SPLINE
SPL {X  -160.000, Y  +499.279, Z    +0.000, E1   +38.981, E3 +82505.209}
SPL {X  -160.000, Y  +490.068, Z    +0.000, E1   +40.198, E3 +82521.513}
SPL {X  -160.000, Y  +481.368, Z    +0.000, E1   +41.274, E3 +82536.503}
SPL {X  -160.000, Y  +470.910, Z    +0.000, E1   +42.658, E3 +82553.012}
SPL {X  -160.000, Y  +460.219, Z    +0.000, E1   +43.912, E3 +82569.633}
SPL {X  -160.000, Y  +451.951, Z    +0.000, E1   +44.355, E3 +82585.198}
SPL {X  -160.000, Y  +442.331, Z    +0.000, E1   +44.390, E3 +82606.062}
SPL {X  -160.000, Y  +433.037, Z    +0.000, E1   +44.348, E3 +82626.336}
SPL {X  -160.000, Y  +424.435, Z    +0.000, E1   +44.358, E3 +82645.005}
SPL {X  -160.000, Y  +416.015, Z    +0.000, E1   +44.348, E3 +82663.325}
SPL {X  -160.000, Y  +407.167, Z    +0.000, E1   +44.365, E3 +82682.535}
SPL {X  -160.000, Y  +397.599, Z    +0.000, E1   +44.371, E3 +82703.344}
SPL {X  -160.000, Y  +388.533, Z    +0.000, E1   +44.340, E3 +82723.119}
SPL {X  -159.759, Y  +380.021, Z    +0.000, E1   +44.311, E3 +82741.851}
SPL {X  -159.014, Y  +371.065, Z    +0.000, E1   +44.193, E3 +82762.089}
SPL {X  -157.745, Y  +362.030, Z    +0.000, E1   +43.965, E3 +82783.071}
SPL {X  -156.258, Y  +354.400, Z    +0.000, E1   +43.653, E3 +82801.278}
SPL {X  -154.385, Y  +346.786, Z    +0.000, E1   +43.356, E3 +82819.690}
SPL {X  -152.146, Y  +339.286, Z    +0.000, E1   +42.904, E3 +82838.324}
SPL {X  -149.854, Y  +332.731, Z    +0.000, E1   +42.474, E3 +82854.852}
SPL {X  -145.635, Y  +322.541, Z    +0.000, E1   +36.397, E3 +82930.811}
ENDSPLINE

SPLINE
SPL {X  -156.682, Y  +356.385, Z    +0.000, E1   +19.033, E3 +82989.117}
SPL {X  -159.526, Y  +376.492, Z    +0.000, E1    +8.067, E3 +82999.026}
SPL {X  -159.961, Y  +385.275, Z    +0.000, E1    +2.550, E3 +83001.065}
SPL {X  -160.000, Y  +390.345, Z    +0.000, E1    -1.188, E3 +83001.791}
SPL {X  -160.000, Y  +395.838, Z    +0.000, E1    -6.211, E3 +83002.734}
SPL {X  -160.000, Y  +403.277, Z    +0.000, E1   -14.057, E3 +83004.685}
SPL {X  -160.000, Y  +414.316, Z    +0.000, E1   -24.810, E3 +83009.758}
SPL {X  -160.000, Y  +442.604, Z    +0.000, E1   -40.161, E3 +83031.893}
SPL {X  -160.000, Y  +482.867, Z    +0.000, E1   -45.148, E3 +83092.109}
SPL {X  -160.000, Y  +494.769, Z    +0.000, E1   -45.151, E3 +83117.328}
SPL {X  -160.000, Y  +505.761, Z    +0.000, E1   -45.118, E3 +83140.642}
SPL {X  -160.000, Y  +517.347, Z    +0.000, E1   -45.173, E3 +83165.080}
SPL {X  -160.000, Y  +529.298, Z    +0.000, E1   -45.138, E3 +83190.463}
SPL {X  -160.000, Y  +540.664, Z    +0.000, E1   -45.139, E3 +83214.541}
SPL {X  -160.000, Y  +552.011, Z    +0.000, E1   -45.139, E3 +83238.577}
SPL {X  -160.000, Y  +563.667, Z    +0.000, E1   -45.146, E3 +83263.257}
SPL {X  -160.000, Y  +574.965, Z    +0.000, E1   -45.125, E3 +83287.233}
SPL {X  -160.000, Y  +585.644, Z    +0.000, E1   -45.117, E3 +83309.873}
SPL {X  -160.000, Y  +596.819, Z    +0.000, E1   -45.144, E3 +83333.514}
SPL {X  -160.000, Y  +608.165, Z    +0.000, E1   -45.120, E3 +83357.589}
SPL {X  -160.000, Y  +619.270, Z    +0.000, E1   -45.132, E3 +83381.091}
SPL {X  -160.000, Y  +629.968, Z    +0.000, E1   -45.117, E3 +83403.758}
SPL {X  -160.000, Y  +640.750, Z    +0.000, E1   -45.131, E3 +83426.581}
SPL {X  -160.000, Y  +651.429, Z    +0.000, E1   -45.117, E3 +83449.222}
SPL {X  -160.000, Y  +662.434, Z    +0.000, E1   -45.129, E3 +83472.566}
SPL {X  -159.992, Y  +673.110, Z    +0.000, E1   -45.097, E3 +83495.258}
SPL {X  -159.521, Y  +683.874, Z    +0.000, E1   -45.054, E3 +83518.514}
SPL {X  -158.435, Y  +693.823, Z    +0.000, E1   -44.810, E3 +83540.818}
SPL {X  -156.807, Y  +703.304, Z    +0.000, E1   -44.558, E3 +83562.539}
SPL {X  -154.802, Y  +711.950, Z    +0.000, E1   -44.141, E3 +83582.999}
SPL {X  -152.641, Y  +719.464, Z    +0.000, E1   -43.749, E3 +83601.114}
SPL {X  -149.826, Y  +727.645, Z    +0.000, E1   -43.252, E3 +83621.217}
SPL {X  -145.307, Y  +738.478, Z    +0.000, E1   -36.676, E3 +83701.285}
ENDSPLINE

SPLINE
SPL {X  -155.601, Y  +708.762, Z    +0.000, E1   -21.463, E3 +83756.072}
SPL {X  -158.549, Y  +693.002, Z    +0.000, E1   -13.406, E3 +83765.062}
SPL {X  -159.716, Y  +681.031, Z    +0.000, E1    -6.529, E3 +83769.212}
SPL {X  -160.000, Y  +671.641, Z    +0.000, E1    -0.547, E3 +83770.929}
SPL {X  -160.000, Y  +665.424, Z    +0.000, E1    +5.044, E3 +83771.877}
SPL {X  -160.000, Y  +658.015, Z    +0.000, E1   +12.630, E3 +83773.795}
SPL {X  -160.000, Y  +645.110, Z    +0.000, E1   +25.142, E3 +83779.595}
SPL {X  -160.000, Y  +611.664, Z    +0.000, E1   +41.262, E3 +83809.324}
SPL {X  -160.000, Y  +581.433, Z    +0.000, E1   +44.103, E3 +83859.061}
SPL {X  -160.000, Y  +572.090, Z    +0.000, E1   +44.120, E3 +83879.526}
SPL {X  -160.000, Y  +563.431, Z    +0.000, E1   +44.084, E3 +83898.579}
SPL {X  -160.000, Y  +556.107, Z    +0.000, E1   +44.076, E3 +83914.647}
SPL {X  -160.000, Y  +549.181, Z    +0.000, E1   +44.079, E3 +83929.807}
SPL {X  -160.000, Y  +542.413, Z    +0.000, E1   +44.088, E3 +83944.641}
SPL {X  -160.000, Y  +534.609, Z    +0.000, E1   +44.095, E3 +83961.751}
SPL {X  -160.000, Y  +527.457, Z    +0.000, E1   +44.070, E3 +83977.461}
SPL {X  -160.000, Y  +520.912, Z    +0.000, E1   +44.079, E3 +83991.802}
SPL {X  -160.000, Y  +514.086, Z    +0.000, E1   +44.081, E3 +84006.750}
SPL {X  -160.000, Y  +507.208, Z    +0.000, E1   +44.082, E3 +84021.827}
SPL {X  -160.000, Y  +499.184, Z    +0.000, E1   +44.113, E3 +84039.385}
ENDSPLINE

SPLINE
SPL {X  -160.000, Y  +503.824, Z    +0.000, E1   +39.488, E3 +84055.434}
ENDSPLINE

SPLINE
SPL {X  -160.000, Y  +499.279, Z    +0.000, E1   +38.981, E3 +84070.424}
SPL {X  -160.000, Y  +490.068, Z    +0.000, E1   +40.198, E3 +84086.728}
SPL {X  -160.000, Y  +481.368, Z    +0.000, E1   +41.274, E3 +84101.717}
SPL {X  -160.000, Y  +470.910, Z    +0.000, E1   +42.658, E3 +84118.226}
SPL {X  -160.000, Y  +460.219, Z    +0.000, E1   +43.912, E3 +84134.847}
SPL {X  -160.000, Y  +451.951, Z    +0.000, E1   +44.355, E3 +84150.412}
SPL {X  -160.000, Y  +442.331, Z    +0.000, E1   +44.390, E3 +84171.276}
SPL {X  -160.000, Y  +433.037, Z    +0.000, E1   +44.348, E3 +84191.550}
SPL {X  -160.000, Y  +424.435, Z    +0.000, E1   +44.358, E3 +84210.219}
SPL {X  -160.000, Y  +416.015, Z    +0.000, E1   +44.348, E3 +84228.539}
SPL {X  -160.000, Y  +407.167, Z    +0.000, E1   +44.365, E3 +84247.750}
SPL {X  -160.000, Y  +397.599, Z    +0.000, E1   +44.371, E3 +84268.558}
SPL {X  -160.000, Y  +388.533, Z    +0.000, E1   +44.340, E3 +84288.333}
SPL {X  -159.759, Y  +380.021, Z    +0.000, E1   +44.311, E3 +84307.065}
SPL {X  -159.014, Y  +371.065, Z    +0.000, E1   +44.193, E3 +84327.303}
SPL {X  -157.745, Y  +362.030, Z    +0.000, E1   +43.965, E3 +84348.285}
SPL {X  -156.258, Y  +354.400, Z    +0.000, E1   +43.653, E3 +84366.492}
SPL {X  -154.385, Y  +346.786, Z    +0.000, E1   +43.356, E3 +84384.904}
SPL {X  -152.146, Y  +339.286, Z    +0.000, E1   +42.904, E3 +84403.539}
SPL {X  -149.854, Y  +332.731, Z    +0.000, E1   +42.474, E3 +84420.066}
SPL {X  -145.635, Y  +322.541, Z    +0.000, E1   +36.397, E3 +84496.025}
ENDSPLINE

SPLINE
SPL {X  -156.682, Y  +356.385, Z    +0.000, E1   +19.033, E3 +84554.331}
SPL {X  -159.526, Y  +376.492, Z    +0.000, E1    +8.067, E3 +84564.241}
SPL {X  -159.961, Y  +385.275, Z    +0.000, E1    +2.550, E3 +84566.279}
SPL {X  -160.000, Y  +390.345, Z    +0.000, E1    -1.188, E3 +84567.005}
SPL {X  -160.000, Y  +395.838, Z    +0.000, E1    -6.211, E3 +84567.948}
SPL {X  -160.000, Y  +403.277, Z    +0.000, E1   -14.057, E3 +84569.900}
SPL {X  -160.000, Y  +414.316, Z    +0.000, E1   -24.810, E3 +84574.973}
SPL {X  -160.000, Y  +442.604, Z    +0.000, E1   -40.161, E3 +84597.107}
SPL {X  -160.000, Y  +482.867, Z    +0.000, E1   -45.148, E3 +84657.323}
SPL {X  -160.000, Y  +494.769, Z    +0.000, E1   -45.151, E3 +84682.542}
SPL {X  -160.000, Y  +505.761, Z    +0.000, E1   -45.118, E3 +84705.856}
SPL {X  -160.000, Y  +517.347, Z    +0.000, E1   -45.173, E3 +84730.294}
SPL {X  -160.000, Y  +529.298, Z    +0.000, E1   -45.138, E3 +84755.677}
SPL {X  -160.000, Y  +540.664, Z    +0.000, E1   -45.139, E3 +84779.755}
SPL {X  -160.000, Y  +552.011, Z    +0.000, E1   -45.139, E3 +84803.791}
SPL {X  -160.000, Y  +563.667, Z    +0.000, E1   -45.146, E3 +84828.471}
SPL {X  -160.000, Y  +574.965, Z    +0.000, E1   -45.125, E3 +84852.447}
SPL {X  -160.000, Y  +585.644, Z    +0.000, E1   -45.117, E3 +84875.087}
SPL {X  -160.000, Y  +596.819, Z    +0.000, E1   -45.144, E3 +84898.729}
SPL {X  -160.000, Y  +608.165, Z    +0.000, E1   -45.120, E3 +84922.803}
SPL {X  -160.000, Y  +619.270, Z    +0.000, E1   -45.132, E3 +84946.305}
SPL {X  -160.000, Y  +629.968, Z    +0.000, E1   -45.117, E3 +84968.972}
SPL {X  -160.000, Y  +640.750, Z    +0.000, E1   -45.131, E3 +84991.795}
SPL {X  -160.000, Y  +651.429, Z    +0.000, E1   -45.117, E3 +85014.436}
SPL {X  -160.000, Y  +662.434, Z    +0.000, E1   -45.129, E3 +85037.780}
SPL {X  -159.992, Y  +673.110, Z    +0.000, E1   -45.097, E3 +85060.473}
SPL {X  -159.521, Y  +683.874, Z    +0.000, E1   -45.054, E3 +85083.728}
SPL {X  -158.435, Y  +693.823, Z    +0.000, E1   -44.810, E3 +85106.032}
SPL {X  -156.807, Y  +703.304, Z    +0.000, E1   -44.558, E3 +85127.753}
SPL {X  -154.802, Y  +711.950, Z    +0.000, E1   -44.141, E3 +85148.213}
SPL {X  -152.641, Y  +719.464, Z    +0.000, E1   -43.749, E3 +85166.329}
SPL {X  -149.826, Y  +727.645, Z    +0.000, E1   -43.252, E3 +85186.431}
SPL {X  -145.307, Y  +738.478, Z    +0.000, E1   -36.676, E3 +85266.499}
ENDSPLINE

SPLINE
SPL {X  -155.601, Y  +708.762, Z    +0.000, E1   -21.463, E3 +85321.286}
SPL {X  -158.549, Y  +693.002, Z    +0.000, E1   -13.406, E3 +85330.276}
SPL {X  -159.716, Y  +681.031, Z    +0.000, E1    -6.529, E3 +85334.427}
SPL {X  -160.000, Y  +671.641, Z    +0.000, E1    -0.547, E3 +85336.143}
SPL {X  -160.000, Y  +665.424, Z    +0.000, E1    +5.044, E3 +85337.091}
SPL {X  -160.000, Y  +658.015, Z    +0.000, E1   +12.630, E3 +85339.009}
SPL {X  -160.000, Y  +645.110, Z    +0.000, E1   +25.142, E3 +85344.809}
SPL {X  -160.000, Y  +611.664, Z    +0.000, E1   +41.262, E3 +85374.539}
SPL {X  -160.000, Y  +581.433, Z    +0.000, E1   +44.103, E3 +85424.275}
SPL {X  -160.000, Y  +572.090, Z    +0.000, E1   +44.120, E3 +85444.740}
SPL {X  -160.000, Y  +563.431, Z    +0.000, E1   +44.084, E3 +85463.793}
SPL {X  -160.000, Y  +556.107, Z    +0.000, E1   +44.076, E3 +85479.861}
SPL {X  -160.000, Y  +549.181, Z    +0.000, E1   +44.079, E3 +85495.021}
SPL {X  -160.000, Y  +542.413, Z    +0.000, E1   +44.088, E3 +85509.855}
SPL {X  -160.000, Y  +534.609, Z    +0.000, E1   +44.095, E3 +85526.965}
SPL {X  -160.000, Y  +527.457, Z    +0.000, E1   +44.070, E3 +85542.675}
SPL {X  -160.000, Y  +520.912, Z    +0.000, E1   +44.079, E3 +85557.016}
SPL {X  -160.000, Y  +514.086, Z    +0.000, E1   +44.081, E3 +85571.964}
SPL {X  -160.000, Y  +507.208, Z    +0.000, E1   +44.082, E3 +85587.041}
SPL {X  -160.000, Y  +499.184, Z    +0.000, E1   +44.113, E3 +85604.599}
ENDSPLINE

SPLINE
SPL {X  -160.000, Y  +503.824, Z    +0.000, E1   +39.488, E3 +85620.648}
ENDSPLINE

SPLINE
SPL {X  -160.000, Y  +499.279, Z    +0.000, E1   +38.981, E3 +85635.638}
SPL {X  -160.000, Y  +490.068, Z    +0.000, E1   +40.198, E3 +85651.942}
SPL {X  -160.000, Y  +481.368, Z    +0.000, E1   +41.274, E3 +85666.932}
SPL {X  -160.000, Y  +470.910, Z    +0.000, E1   +42.658, E3 +85683.440}
SPL {X  -160.000, Y  +460.219, Z    +0.000, E1   +43.912, E3 +85700.061}
SPL {X  -160.000, Y  +451.951, Z    +0.000, E1   +44.355, E3 +85715.626}
SPL {X  -160.000, Y  +442.331, Z    +0.000, E1   +44.390, E3 +85736.491}
SPL {X  -160.000, Y  +433.037, Z    +0.000, E1   +44.348, E3 +85756.765}
SPL {X  -160.000, Y  +424.435, Z    +0.000, E1   +44.358, E3 +85775.433}
SPL {X  -160.000, Y  +416.015, Z    +0.000, E1   +44.348, E3 +85793.753}
SPL {X  -160.000, Y  +407.167, Z    +0.000, E1   +44.365, E3 +85812.964}
SPL {X  -160.000, Y  +397.599, Z    +0.000, E1   +44.371, E3 +85833.772}
SPL {X  -160.000, Y  +388.533, Z    +0.000, E1   +44.340, E3 +85853.547}
SPL {X  -159.759, Y  +380.021, Z    +0.000, E1   +44.311, E3 +85872.279}
SPL {X  -159.014, Y  +371.065, Z    +0.000, E1   +44.193, E3 +85892.517}
SPL {X  -157.745, Y  +362.030, Z    +0.000, E1   +43.965, E3 +85913.499}
SPL {X  -156.258, Y  +354.400, Z    +0.000, E1   +43.653, E3 +85931.706}
SPL {X  -154.385, Y  +346.786, Z    +0.000, E1   +43.356, E3 +85950.118}
SPL {X  -152.146, Y  +339.286, Z    +0.000, E1   +42.904, E3 +85968.753}
SPL {X  -149.854, Y  +332.731, Z    +0.000, E1   +42.474, E3 +85985.281}
SPL {X  -145.635, Y  +322.541, Z    +0.000, E1   +36.397, E3 +86061.240}
ENDSPLINE

SPLINE
SPL {X  -156.682, Y  +356.385, Z    +0.000, E1   +19.033, E3 +86119.546}
SPL {X  -159.526, Y  +376.492, Z    +0.000, E1    +8.067, E3 +86129.455}
SPL {X  -159.961, Y  +385.275, Z    +0.000, E1    +2.550, E3 +86131.493}
SPL {X  -160.000, Y  +390.345, Z    +0.000, E1    -1.188, E3 +86132.219}
SPL {X  -160.000, Y  +395.838, Z    +0.000, E1    -6.211, E3 +86133.163}
SPL {X  -160.000, Y  +403.277, Z    +0.000, E1   -14.057, E3 +86135.114}
SPL {X  -160.000, Y  +414.316, Z    +0.000, E1   -24.810, E3 +86140.187}
SPL {X  -160.000, Y  +442.604, Z    +0.000, E1   -40.161, E3 +86162.321}
SPL {X  -160.000, Y  +482.867, Z    +0.000, E1   -45.148, E3 +86222.537}
SPL {X  -160.000, Y  +494.769, Z    +0.000, E1   -45.151, E3 +86247.756}
SPL {X  -160.000, Y  +505.761, Z    +0.000, E1   -45.118, E3 +86271.070}
SPL {X  -160.000, Y  +517.347, Z    +0.000, E1   -45.173, E3 +86295.508}
SPL {X  -160.000, Y  +529.298, Z    +0.000, E1   -45.138, E3 +86320.891}
SPL {X  -160.000, Y  +540.664, Z    +0.000, E1   -45.139, E3 +86344.969}
SPL {X  -160.000, Y  +552.011, Z    +0.000, E1   -45.139, E3 +86369.005}
SPL {X  -160.000, Y  +563.667, Z    +0.000, E1   -45.146, E3 +86393.685}
SPL {X  -160.000, Y  +574.965, Z    +0.000, E1   -45.125, E3 +86417.661}
SPL {X  -160.000, Y  +585.644, Z    +0.000, E1   -45.117, E3 +86440.301}
SPL {X  -160.000, Y  +596.819, Z    +0.000, E1   -45.144, E3 +86463.943}
SPL {X  -160.000, Y  +608.165, Z    +0.000, E1   -45.120, E3 +86488.017}
SPL {X  -160.000, Y  +619.270, Z    +0.000, E1   -45.132, E3 +86511.520}
SPL {X  -160.000, Y  +629.968, Z    +0.000, E1   -45.117, E3 +86534.186}
SPL {X  -160.000, Y  +640.750, Z    +0.000, E1   -45.131, E3 +86557.009}
SPL {X  -160.000, Y  +651.429, Z    +0.000, E1   -45.117, E3 +86579.650}
SPL {X  -160.000, Y  +662.434, Z    +0.000, E1   -45.129, E3 +86602.994}
SPL {X  -159.992, Y  +673.110, Z    +0.000, E1   -45.097, E3 +86625.687}
SPL {X  -159.521, Y  +683.874, Z    +0.000, E1   -45.054, E3 +86648.942}
SPL {X  -158.435, Y  +693.823, Z    +0.000, E1   -44.810, E3 +86671.246}
SPL {X  -156.807, Y  +703.304, Z    +0.000, E1   -44.558, E3 +86692.967}
SPL {X  -154.802, Y  +711.950, Z    +0.000, E1   -44.141, E3 +86713.427}
SPL {X  -152.641, Y  +719.464, Z    +0.000, E1   -43.749, E3 +86731.543}
SPL {X  -149.826, Y  +727.645, Z    +0.000, E1   -43.252, E3 +86751.646}
SPL {X  -145.307, Y  +738.478, Z    +0.000, E1   -36.676, E3 +86831.713}
ENDSPLINE

SPLINE
SPL {X  -155.601, Y  +708.762, Z    +0.000, E1   -21.463, E3 +86886.500}
SPL {X  -158.549, Y  +693.002, Z    +0.000, E1   -13.406, E3 +86895.491}
SPL {X  -159.716, Y  +681.031, Z    +0.000, E1    -6.529, E3 +86899.641}
SPL {X  -160.000, Y  +671.641, Z    +0.000, E1    -0.547, E3 +86901.357}
SPL {X  -160.000, Y  +665.424, Z    +0.000, E1    +5.044, E3 +86902.306}
SPL {X  -160.000, Y  +658.015, Z    +0.000, E1   +12.630, E3 +86904.223}
SPL {X  -160.000, Y  +645.110, Z    +0.000, E1   +25.142, E3 +86910.023}
SPL {X  -160.000, Y  +611.664, Z    +0.000, E1   +41.262, E3 +86939.753}
SPL {X  -160.000, Y  +581.433, Z    +0.000, E1   +44.103, E3 +86989.489}
SPL {X  -160.000, Y  +572.090, Z    +0.000, E1   +44.120, E3 +87009.954}
SPL {X  -160.000, Y  +563.431, Z    +0.000, E1   +44.084, E3 +87029.007}
SPL {X  -160.000, Y  +556.107, Z    +0.000, E1   +44.076, E3 +87045.075}
SPL {X  -160.000, Y  +549.181, Z    +0.000, E1   +44.079, E3 +87060.235}
SPL {X  -160.000, Y  +542.413, Z    +0.000, E1   +44.088, E3 +87075.069}
SPL {X  -160.000, Y  +534.609, Z    +0.000, E1   +44.095, E3 +87092.179}
SPL {X  -160.000, Y  +527.457, Z    +0.000, E1   +44.070, E3 +87107.889}
SPL {X  -160.000, Y  +520.912, Z    +0.000, E1   +44.079, E3 +87122.230}
SPL {X  -160.000, Y  +514.086, Z    +0.000, E1   +44.081, E3 +87137.179}
SPL {X  -160.000, Y  +507.208, Z    +0.000, E1   +44.082, E3 +87152.255}
SPL {X  -160.000, Y  +499.184, Z    +0.000, E1   +44.113, E3 +87169.813}
ENDSPLINE

SPLINE
SPL {X  -160.000, Y  +503.824, Z    +0.000, E1   +39.488, E3 +87185.862}
ENDSPLINE

SPLINE
SPL {X  -160.000, Y  +499.279, Z    +0.000, E1   +38.981, E3 +87200.852}
SPL {X  -160.000, Y  +490.068, Z    +0.000, E1   +40.198, E3 +87217.156}
SPL {X  -160.000, Y  +481.368, Z    +0.000, E1   +41.274, E3 +87232.146}
SPL {X  -160.000, Y  +470.910, Z    +0.000, E1   +42.658, E3 +87248.654}
SPL {X  -160.000, Y  +460.219, Z    +0.000, E1   +43.912, E3 +87265.275}
SPL {X  -160.000, Y  +451.951, Z    +0.000, E1   +44.355, E3 +87280.841}
SPL {X  -160.000, Y  +442.331, Z    +0.000, E1   +44.390, E3 +87301.705}
SPL {X  -160.000, Y  +433.037, Z    +0.000, E1   +44.348, E3 +87321.979}
SPL {X  -160.000, Y  +424.435, Z    +0.000, E1   +44.358, E3 +87340.647}
SPL {X  -160.000, Y  +416.015, Z    +0.000, E1   +44.348, E3 +87358.967}
SPL {X  -160.000, Y  +407.167, Z    +0.000, E1   +44.365, E3 +87378.178}
SPL {X  -160.000, Y  +397.599, Z    +0.000, E1   +44.371, E3 +87398.986}
SPL {X  -160.000, Y  +388.533, Z    +0.000, E1   +44.340, E3 +87418.761}
SPL {X  -159.759, Y  +380.021, Z    +0.000, E1   +44.311, E3 +87437.493}
SPL {X  -159.014, Y  +371.065, Z    +0.000, E1   +44.193, E3 +87457.731}
SPL {X  -157.745, Y  +362.030, Z    +0.000, E1   +43.965, E3 +87478.713}
SPL {X  -156.258, Y  +354.400, Z    +0.000, E1   +43.653, E3 +87496.921}
SPL {X  -154.385, Y  +346.786, Z    +0.000, E1   +43.356, E3 +87515.332}
SPL {X  -152.146, Y  +339.286, Z    +0.000, E1   +42.904, E3 +87533.967}
SPL {X  -149.854, Y  +332.731, Z    +0.000, E1   +42.474, E3 +87550.495}
SPL {X  -145.635, Y  +322.541, Z    +0.000, E1   +36.397, E3 +87626.454}
ENDSPLINE

SPLINE
SPL {X  -156.682, Y  +356.385, Z    +0.000, E1   +19.033, E3 +87684.760}
SPL {X  -159.526, Y  +376.492, Z    +0.000, E1    +8.067, E3 +87694.669}
SPL {X  -159.961, Y  +385.275, Z    +0.000, E1    +2.550, E3 +87696.707}
SPL {X  -160.000, Y  +390.345, Z    +0.000, E1    -1.188, E3 +87697.433}
SPL {X  -160.000, Y  +395.838, Z    +0.000, E1    -6.211, E3 +87698.377}
SPL {X  -160.000, Y  +403.277, Z    +0.000, E1   -14.057, E3 +87700.328}
SPL {X  -160.000, Y  +414.316, Z    +0.000, E1   -24.810, E3 +87705.401}
SPL {X  -160.000, Y  +442.604, Z    +0.000, E1   -40.161, E3 +87727.535}
SPL {X  -160.000, Y  +482.867, Z    +0.000, E1   -45.148, E3 +87787.751}
SPL {X  -160.000, Y  +494.769, Z    +0.000, E1   -45.151, E3 +87812.971}
SPL {X  -160.000, Y  +505.761, Z    +0.000, E1   -45.118, E3 +87836.284}
SPL {X  -160.000, Y  +517.347, Z    +0.000, E1   -45.173, E3 +87860.722}
SPL {X  -160.000, Y  +529.298, Z    +0.000, E1   -45.138, E3 +87886.105}
SPL {X  -160.000, Y  +540.664, Z    +0.000, E1   -45.139, E3 +87910.183}
SPL {X  -160.000, Y  +552.011, Z    +0.000, E1   -45.139, E3 +87934.219}
SPL {X  -160.000, Y  +563.667, Z    +0.000, E1   -45.146, E3 +87958.900}
SPL {X  -160.000, Y  +574.965, Z    +0.000, E1   -45.125, E3 +87982.875}
SPL {X  -160.000, Y  +585.644, Z    +0.000, E1   -45.117, E3 +88005.515}
SPL {X  -160.000, Y  +596.819, Z    +0.000, E1   -45.144, E3 +88029.157}
SPL {X  -160.000, Y  +608.165, Z    +0.000, E1   -45.120, E3 +88053.231}
SPL {X  -160.000, Y  +619.270, Z    +0.000, E1   -45.132, E3 +88076.734}
SPL {X  -160.000, Y  +629.968, Z    +0.000, E1   -45.117, E3 +88099.400}
SPL {X  -160.000, Y  +640.750, Z    +0.000, E1   -45.131, E3 +88122.223}
SPL {X  -160.000, Y  +651.429, Z    +0.000, E1   -45.117, E3 +88144.864}
SPL {X  -160.000, Y  +662.434, Z    +0.000, E1   -45.129, E3 +88168.208}
SPL {X  -159.992, Y  +673.110, Z    +0.000, E1   -45.097, E3 +88190.901}
SPL {X  -159.521, Y  +683.874, Z    +0.000, E1   -45.054, E3 +88214.156}
SPL {X  -158.435, Y  +693.823, Z    +0.000, E1   -44.810, E3 +88236.460}
SPL {X  -156.807, Y  +703.304, Z    +0.000, E1   -44.558, E3 +88258.181}
SPL {X  -154.802, Y  +711.950, Z    +0.000, E1   -44.141, E3 +88278.641}
SPL {X  -152.641, Y  +719.464, Z    +0.000, E1   -43.749, E3 +88296.757}
SPL {X  -149.826, Y  +727.645, Z    +0.000, E1   -43.252, E3 +88316.860}
SPL {X  -145.307, Y  +738.478, Z    +0.000, E1   -36.676, E3 +88396.927}
ENDSPLINE

SPLINE
SPL {X  -155.601, Y  +708.762, Z    +0.000, E1   -21.463, E3 +88451.714}
SPL {X  -158.549, Y  +693.002, Z    +0.000, E1   -13.406, E3 +88460.705}
SPL {X  -159.716, Y  +681.031, Z    +0.000, E1    -6.529, E3 +88464.855}
SPL {X  -160.000, Y  +671.641, Z    +0.000, E1    -0.547, E3 +88466.571}
SPL {X  -160.000, Y  +665.424, Z    +0.000, E1    +5.044, E3 +88467.520}
SPL {X  -160.000, Y  +658.015, Z    +0.000, E1   +12.630, E3 +88469.437}
SPL {X  -160.000, Y  +645.110, Z    +0.000, E1   +25.142, E3 +88475.238}
SPL {X  -160.000, Y  +611.664, Z    +0.000, E1   +41.262, E3 +88504.967}
SPL {X  -160.000, Y  +581.433, Z    +0.000, E1   +44.103, E3 +88554.704}
SPL {X  -160.000, Y  +572.090, Z    +0.000, E1   +44.120, E3 +88575.168}
SPL {X  -160.000, Y  +563.431, Z    +0.000, E1   +44.084, E3 +88594.221}
SPL {X  -160.000, Y  +556.107, Z    +0.000, E1   +44.076, E3 +88610.290}
SPL {X  -160.000, Y  +549.181, Z    +0.000, E1   +44.079, E3 +88625.449}
SPL {X  -160.000, Y  +542.413, Z    +0.000, E1   +44.088, E3 +88640.283}
SPL {X  -160.000, Y  +534.609, Z    +0.000, E1   +44.095, E3 +88657.393}
SPL {X  -160.000, Y  +527.457, Z    +0.000, E1   +44.070, E3 +88673.104}
SPL {X  -160.000, Y  +520.912, Z    +0.000, E1   +44.079, E3 +88687.444}
SPL {X  -160.000, Y  +514.086, Z    +0.000, E1   +44.081, E3 +88702.393}
SPL {X  -160.000, Y  +507.208, Z    +0.000, E1   +44.082, E3 +88717.469}
SPL {X  -160.000, Y  +499.184, Z    +0.000, E1   +44.113, E3 +88735.027}
ENDSPLINE

SPLINE
SPL {X  -160.000, Y  +503.824, Z    +0.000, E1   +39.488, E3 +88751.076}
ENDSPLINE

SPLINE
SPL {X  -160.000, Y  +499.279, Z    +0.000, E1   +38.981, E3 +88766.066}
SPL {X  -160.000, Y  +490.068, Z    +0.000, E1   +40.198, E3 +88782.370}
SPL {X  -160.000, Y  +481.368, Z    +0.000, E1   +41.274, E3 +88797.360}
SPL {X  -160.000, Y  +470.910, Z    +0.000, E1   +42.658, E3 +88813.869}
SPL {X  -160.000, Y  +460.219, Z    +0.000, E1   +43.912, E3 +88830.489}
SPL {X  -160.000, Y  +451.951, Z    +0.000, E1   +44.355, E3 +88846.055}
SPL {X  -160.000, Y  +442.331, Z    +0.000, E1   +44.390, E3 +88866.919}
SPL {X  -160.000, Y  +433.037, Z    +0.000, E1   +44.348, E3 +88887.193}
SPL {X  -160.000, Y  +424.435, Z    +0.000, E1   +44.358, E3 +88905.861}
SPL {X  -160.000, Y  +416.015, Z    +0.000, E1   +44.348, E3 +88924.181}
SPL {X  -160.000, Y  +407.167, Z    +0.000, E1   +44.365, E3 +88943.392}
SPL {X  -160.000, Y  +397.599, Z    +0.000, E1   +44.371, E3 +88964.200}
SPL {X  -160.000, Y  +388.533, Z    +0.000, E1   +44.340, E3 +88983.975}
SPL {X  -159.759, Y  +380.021, Z    +0.000, E1   +44.311, E3 +89002.707}
SPL {X  -159.014, Y  +371.065, Z    +0.000, E1   +44.193, E3 +89022.945}
SPL {X  -157.745, Y  +362.030, Z    +0.000, E1   +43.965, E3 +89043.927}
SPL {X  -156.258, Y  +354.400, Z    +0.000, E1   +43.653, E3 +89062.135}
SPL {X  -154.385, Y  +346.786, Z    +0.000, E1   +43.356, E3 +89080.547}
SPL {X  -152.146, Y  +339.286, Z    +0.000, E1   +42.904, E3 +89099.181}
SPL {X  -149.854, Y  +332.731, Z    +0.000, E1   +42.474, E3 +89115.709}
SPL {X  -145.635, Y  +322.541, Z    +0.000, E1   +36.397, E3 +89191.668}
ENDSPLINE

SPLINE
SPL {X  -156.682, Y  +356.385, Z    +0.000, E1   +19.033, E3 +89249.974}
SPL {X  -159.526, Y  +376.492, Z    +0.000, E1    +8.067, E3 +89259.883}
SPL {X  -159.961, Y  +385.275, Z    +0.000, E1    +2.550, E3 +89261.921}
SPL {X  -160.000, Y  +390.345, Z    +0.000, E1    -1.188, E3 +89262.647}
SPL {X  -160.000, Y  +395.838, Z    +0.000, E1    -6.211, E3 +89263.591}
SPL {X  -160.000, Y  +403.277, Z    +0.000, E1   -14.057, E3 +89265.542}
SPL {X  -160.000, Y  +414.316, Z    +0.000, E1   -24.810, E3 +89270.615}
SPL {X  -160.000, Y  +442.604, Z    +0.000, E1   -40.161, E3 +89292.749}
SPL {X  -160.000, Y  +482.867, Z    +0.000, E1   -45.148, E3 +89352.965}
SPL {X  -160.000, Y  +494.769, Z    +0.000, E1   -45.151, E3 +89378.185}
SPL {X  -160.000, Y  +505.761, Z    +0.000, E1   -45.118, E3 +89401.499}
SPL {X  -160.000, Y  +517.347, Z    +0.000, E1   -45.173, E3 +89425.936}
SPL {X  -160.000, Y  +529.298, Z    +0.000, E1   -45.138, E3 +89451.320}
SPL {X  -160.000, Y  +540.664, Z    +0.000, E1   -45.139, E3 +89475.398}
SPL {X  -160.000, Y  +552.011, Z    +0.000, E1   -45.139, E3 +89499.433}
SPL {X  -160.000, Y  +563.667, Z    +0.000, E1   -45.146, E3 +89524.114}
SPL {X  -160.000, Y  +574.965, Z    +0.000, E1   -45.125, E3 +89548.089}
SPL {X  -160.000, Y  +585.644, Z    +0.000, E1   -45.117, E3 +89570.729}
SPL {X  -160.000, Y  +596.819, Z    +0.000, E1   -45.144, E3 +89594.371}
SPL {X  -160.000, Y  +608.165, Z    +0.000, E1   -45.120, E3 +89618.445}
SPL {X  -160.000, Y  +619.270, Z    +0.000, E1   -45.132, E3 +89641.948}
SPL {X  -160.000, Y  +629.968, Z    +0.000, E1   -45.117, E3 +89664.614}
SPL {X  -160.000, Y  +640.750, Z    +0.000, E1   -45.131, E3 +89687.437}
SPL {X  -160.000, Y  +651.429, Z    +0.000, E1   -45.117, E3 +89710.078}
SPL {X  -160.000, Y  +662.434, Z    +0.000, E1   -45.129, E3 +89733.422}
SPL {X  -159.992, Y  +673.110, Z    +0.000, E1   -45.097, E3 +89756.115}
SPL {X  -159.521, Y  +683.874, Z    +0.000, E1   -45.054, E3 +89779.370}
SPL {X  -158.435, Y  +693.823, Z    +0.000, E1   -44.810, E3 +89801.674}
SPL {X  -156.807, Y  +703.304, Z    +0.000, E1   -44.558, E3 +89823.395}
SPL {X  -154.802, Y  +711.950, Z    +0.000, E1   -44.141, E3 +89843.855}
SPL {X  -152.641, Y  +719.464, Z    +0.000, E1   -43.749, E3 +89861.971}
SPL {X  -149.826, Y  +727.645, Z    +0.000, E1   -43.252, E3 +89882.074}
SPL {X  -145.307, Y  +738.478, Z    +0.000, E1   -36.676, E3 +89962.141}
ENDSPLINE

SPLINE
SPL {X  -155.601, Y  +708.762, Z    +0.000, E1   -21.463, E3 +90016.928}
SPL {X  -158.549, Y  +693.002, Z    +0.000, E1   -13.406, E3 +90025.919}
SPL {X  -159.716, Y  +681.031, Z    +0.000, E1    -6.529, E3 +90030.069}
SPL {X  -160.000, Y  +671.641, Z    +0.000, E1    -0.547, E3 +90031.786}
SPL {X  -160.000, Y  +665.424, Z    +0.000, E1    +5.044, E3 +90032.734}
SPL {X  -160.000, Y  +658.015, Z    +0.000, E1   +12.630, E3 +90034.652}
SPL {X  -160.000, Y  +645.110, Z    +0.000, E1   +25.142, E3 +90040.452}
SPL {X  -160.000, Y  +611.664, Z    +0.000, E1   +41.262, E3 +90070.181}
SPL {X  -160.000, Y  +581.433, Z    +0.000, E1   +44.103, E3 +90119.918}
SPL {X  -160.000, Y  +572.090, Z    +0.000, E1   +44.120, E3 +90140.382}
SPL {X  -160.000, Y  +563.431, Z    +0.000, E1   +44.084, E3 +90159.435}
SPL {X  -160.000, Y  +556.107, Z    +0.000, E1   +44.076, E3 +90175.504}
SPL {X  -160.000, Y  +549.181, Z    +0.000, E1   +44.079, E3 +90190.663}
SPL {X  -160.000, Y  +542.413, Z    +0.000, E1   +44.088, E3 +90205.497}
SPL {X  -160.000, Y  +534.609, Z    +0.000, E1   +44.095, E3 +90222.607}
SPL {X  -160.000, Y  +527.457, Z    +0.000, E1   +44.070, E3 +90238.318}
SPL {X  -160.000, Y  +520.912, Z    +0.000, E1   +44.079, E3 +90252.659}
SPL {X  -160.000, Y  +514.086, Z    +0.000, E1   +44.081, E3 +90267.607}
SPL {X  -160.000, Y  +507.208, Z    +0.000, E1   +44.082, E3 +90282.683}
SPL {X  -160.000, Y  +499.184, Z    +0.000, E1   +44.113, E3 +90300.241}
ENDSPLINE

SPLINE
SPL {X  -160.000, Y  +503.824, Z    +0.000, E1   +39.488, E3 +90316.290}
ENDSPLINE

SPLINE
SPL {X  -160.000, Y  +499.279, Z    +0.000, E1   +38.981, E3 +90331.280}
SPL {X  -160.000, Y  +490.068, Z    +0.000, E1   +40.198, E3 +90347.584}
SPL {X  -160.000, Y  +481.368, Z    +0.000, E1   +41.274, E3 +90362.574}
SPL {X  -160.000, Y  +470.910, Z    +0.000, E1   +42.658, E3 +90379.083}
SPL {X  -160.000, Y  +460.219, Z    +0.000, E1   +43.912, E3 +90395.703}
SPL {X  -160.000, Y  +451.951, Z    +0.000, E1   +44.355, E3 +90411.269}
SPL {X  -160.000, Y  +442.331, Z    +0.000, E1   +44.390, E3 +90432.133}
SPL {X  -160.000, Y  +433.037, Z    +0.000, E1   +44.348, E3 +90452.407}
SPL {X  -160.000, Y  +424.435, Z    +0.000, E1   +44.358, E3 +90471.075}
SPL {X  -160.000, Y  +416.015, Z    +0.000, E1   +44.348, E3 +90489.395}
SPL {X  -160.000, Y  +407.167, Z    +0.000, E1   +44.365, E3 +90508.606}
SPL {X  -160.000, Y  +397.599, Z    +0.000, E1   +44.371, E3 +90529.415}
SPL {X  -160.000, Y  +388.533, Z    +0.000, E1   +44.340, E3 +90549.189}
SPL {X  -159.759, Y  +380.021, Z    +0.000, E1   +44.311, E3 +90567.921}
SPL {X  -159.014, Y  +371.065, Z    +0.000, E1   +44.193, E3 +90588.160}
SPL {X  -157.745, Y  +362.030, Z    +0.000, E1   +43.965, E3 +90609.141}
SPL {X  -156.258, Y  +354.400, Z    +0.000, E1   +43.653, E3 +90627.349}
SPL {X  -154.385, Y  +346.786, Z    +0.000, E1   +43.356, E3 +90645.761}
SPL {X  -152.146, Y  +339.286, Z    +0.000, E1   +42.904, E3 +90664.395}
SPL {X  -149.854, Y  +332.731, Z    +0.000, E1   +42.474, E3 +90680.923}
SPL {X  -145.635, Y  +322.541, Z    +0.000, E1   +36.397, E3 +90756.882}
ENDSPLINE

SPLINE
SPL {X  -156.682, Y  +356.385, Z    +0.000, E1   +19.033, E3 +90815.188}
SPL {X  -159.526, Y  +376.492, Z    +0.000, E1    +8.067, E3 +90825.097}
SPL {X  -159.961, Y  +385.275, Z    +0.000, E1    +2.550, E3 +90827.136}
SPL {X  -160.000, Y  +390.345, Z    +0.000, E1    -1.188, E3 +90827.862}
SPL {X  -160.000, Y  +395.838, Z    +0.000, E1    -6.211, E3 +90828.805}
SPL {X  -160.000, Y  +403.277, Z    +0.000, E1   -14.057, E3 +90830.756}
SPL {X  -160.000, Y  +414.316, Z    +0.000, E1   -24.810, E3 +90835.829}
SPL {X  -160.000, Y  +442.604, Z    +0.000, E1   -40.161, E3 +90857.963}
SPL {X  -160.000, Y  +482.867, Z    +0.000, E1   -45.148, E3 +90918.180}
SPL {X  -160.000, Y  +494.769, Z    +0.000, E1   -45.151, E3 +90943.399}
SPL {X  -160.000, Y  +505.761, Z    +0.000, E1   -45.118, E3 +90966.713}
SPL {X  -160.000, Y  +517.347, Z    +0.000, E1   -45.173, E3 +90991.150}
SPL {X  -160.000, Y  +529.298, Z    +0.000, E1   -45.138, E3 +91016.534}
SPL {X  -160.000, Y  +540.664, Z    +0.000, E1   -45.139, E3 +91040.612}
SPL {X  -160.000, Y  +552.011, Z    +0.000, E1   -45.139, E3 +91064.648}
SPL {X  -160.000, Y  +563.667, Z    +0.000, E1   -45.146, E3 +91089.328}
SPL {X  -160.000, Y  +574.965, Z    +0.000, E1   -45.125, E3 +91113.304}
SPL {X  -160.000, Y  +585.644, Z    +0.000, E1   -45.117, E3 +91135.944}
SPL {X  -160.000, Y  +596.819, Z    +0.000, E1   -45.144, E3 +91159.585}
SPL {X  -160.000, Y  +608.165, Z    +0.000, E1   -45.120, E3 +91183.659}
SPL {X  -160.000, Y  +619.270, Z    +0.000, E1   -45.132, E3 +91207.162}
SPL {X  -160.000, Y  +629.968, Z    +0.000, E1   -45.117, E3 +91229.828}
SPL {X  -160.000, Y  +640.750, Z    +0.000, E1   -45.131, E3 +91252.651}
SPL {X  -160.000, Y  +651.429, Z    +0.000, E1   -45.117, E3 +91275.293}
SPL {X  -160.000, Y  +662.434, Z    +0.000, E1   -45.129, E3 +91298.637}
SPL {X  -159.992, Y  +673.110, Z    +0.000, E1   -45.097, E3 +91321.329}
SPL {X  -159.521, Y  +683.874, Z    +0.000, E1   -45.054, E3 +91344.584}
SPL {X  -158.435, Y  +693.823, Z    +0.000, E1   -44.810, E3 +91366.889}
SPL {X  -156.807, Y  +703.304, Z    +0.000, E1   -44.558, E3 +91388.609}
SPL {X  -154.802, Y  +711.950, Z    +0.000, E1   -44.141, E3 +91409.069}
SPL {X  -152.641, Y  +719.464, Z    +0.000, E1   -43.749, E3 +91427.185}
SPL {X  -149.826, Y  +727.645, Z    +0.000, E1   -43.252, E3 +91447.288}
SPL {X  -145.307, Y  +738.478, Z    +0.000, E1   -36.676, E3 +91527.356}
ENDSPLINE

SPLINE
SPL {X  -155.601, Y  +708.762, Z    +0.000, E1   -21.463, E3 +91582.142}
SPL {X  -158.549, Y  +693.002, Z    +0.000, E1   -13.406, E3 +91591.133}
SPL {X  -159.716, Y  +681.031, Z    +0.000, E1    -6.529, E3 +91595.283}
SPL {X  -160.000, Y  +671.641, Z    +0.000, E1    -0.547, E3 +91597.000}
SPL {X  -160.000, Y  +665.424, Z    +0.000, E1    +5.044, E3 +91597.948}
SPL {X  -160.000, Y  +658.015, Z    +0.000, E1   +12.630, E3 +91599.866}
SPL {X  -160.000, Y  +645.110, Z    +0.000, E1   +25.142, E3 +91605.666}
SPL {X  -160.000, Y  +611.664, Z    +0.000, E1   +41.262, E3 +91635.395}
SPL {X  -160.000, Y  +581.433, Z    +0.000, E1   +44.103, E3 +91685.132}
SPL {X  -160.000, Y  +572.090, Z    +0.000, E1   +44.120, E3 +91705.596}
SPL {X  -160.000, Y  +563.431, Z    +0.000, E1   +44.084, E3 +91724.650}
SPL {X  -160.000, Y  +556.107, Z    +0.000, E1   +44.076, E3 +91740.718}
SPL {X  -160.000, Y  +549.181, Z    +0.000, E1   +44.079, E3 +91755.878}
SPL {X  -160.000, Y  +542.413, Z    +0.000, E1   +44.088, E3 +91770.711}
SPL {X  -160.000, Y  +534.609, Z    +0.000, E1   +44.095, E3 +91787.822}
SPL {X  -160.000, Y  +527.457, Z    +0.000, E1   +44.070, E3 +91803.532}
SPL {X  -160.000, Y  +520.912, Z    +0.000, E1   +44.079, E3 +91817.873}
SPL {X  -160.000, Y  +514.086, Z    +0.000, E1   +44.081, E3 +91832.821}
SPL {X  -160.000, Y  +507.208, Z    +0.000, E1   +44.082, E3 +91847.897}
SPL {X  -160.000, Y  +499.184, Z    +0.000, E1   +44.113, E3 +91865.456}
ENDSPLINE

SPLINE
SPL {X  -160.000, Y  +503.824, Z    +0.000, E1   +39.488, E3 +91881.504}
ENDSPLINE

SPLINE
SPL {X  -160.000, Y  +499.279, Z    +0.000, E1   +38.981, E3 +91896.494}
SPL {X  -160.000, Y  +490.068, Z    +0.000, E1   +40.198, E3 +91912.798}
SPL {X  -160.000, Y  +481.368, Z    +0.000, E1   +41.274, E3 +91927.788}
SPL {X  -160.000, Y  +470.910, Z    +0.000, E1   +42.658, E3 +91944.297}
SPL {X  -160.000, Y  +460.219, Z    +0.000, E1   +43.912, E3 +91960.918}
SPL {X  -160.000, Y  +451.951, Z    +0.000, E1   +44.355, E3 +91976.483}
SPL {X  -160.000, Y  +442.331, Z    +0.000, E1   +44.390, E3 +91997.347}
SPL {X  -160.000, Y  +433.037, Z    +0.000, E1   +44.348, E3 +92017.621}
SPL {X  -160.000, Y  +424.435, Z    +0.000, E1   +44.358, E3 +92036.290}
SPL {X  -160.000, Y  +416.015, Z    +0.000, E1   +44.348, E3 +92054.610}
SPL {X  -160.000, Y  +407.167, Z    +0.000, E1   +44.365, E3 +92073.820}
SPL {X  -160.000, Y  +397.599, Z    +0.000, E1   +44.371, E3 +92094.629}
SPL {X  -160.000, Y  +388.533, Z    +0.000, E1   +44.340, E3 +92114.404}
SPL {X  -159.759, Y  +380.021, Z    +0.000, E1   +44.311, E3 +92133.136}
SPL {X  -159.014, Y  +371.065, Z    +0.000, E1   +44.193, E3 +92153.374}
SPL {X  -157.745, Y  +362.030, Z    +0.000, E1   +43.965, E3 +92174.356}
SPL {X  -156.258, Y  +354.400, Z    +0.000, E1   +43.653, E3 +92192.563}
SPL {X  -154.385, Y  +346.786, Z    +0.000, E1   +43.356, E3 +92210.975}
SPL {X  -152.146, Y  +339.286, Z    +0.000, E1   +42.904, E3 +92229.609}
SPL {X  -149.854, Y  +332.731, Z    +0.000, E1   +42.474, E3 +92246.137}
SPL {X  -145.635, Y  +322.541, Z    +0.000, E1   +36.397, E3 +92322.096}
ENDSPLINE

SPLINE
SPL {X  -156.682, Y  +356.385, Z    +0.000, E1   +19.033, E3 +92380.402}
SPL {X  -159.526, Y  +376.492, Z    +0.000, E1    +8.067, E3 +92390.311}
SPL {X  -159.961, Y  +385.275, Z    +0.000, E1    +2.550, E3 +92392.350}
SPL {X  -160.000, Y  +390.345, Z    +0.000, E1    -1.188, E3 +92393.076}
SPL {X  -160.000, Y  +395.838, Z    +0.000, E1    -6.211, E3 +92394.019}
SPL {X  -160.000, Y  +403.277, Z    +0.000, E1   -14.057, E3 +92395.970}
SPL {X  -160.000, Y  +414.316, Z    +0.000, E1   -24.810, E3 +92401.043}
SPL {X  -160.000, Y  +442.604, Z    +0.000, E1   -40.161, E3 +92423.178}
SPL {X  -160.000, Y  +482.867, Z    +0.000, E1   -45.148, E3 +92483.394}
SPL {X  -160.000, Y  +494.769, Z    +0.000, E1   -45.151, E3 +92508.613}
SPL {X  -160.000, Y  +505.761, Z    +0.000, E1   -45.118, E3 +92531.927}
SPL {X  -160.000, Y  +517.347, Z    +0.000, E1   -45.173, E3 +92556.365}
SPL {X  -160.000, Y  +529.298, Z    +0.000, E1   -45.138, E3 +92581.748}
SPL {X  -160.000, Y  +540.664, Z    +0.000, E1   -45.139, E3 +92605.826}
SPL {X  -160.000, Y  +552.011, Z    +0.000, E1   -45.139, E3 +92629.862}
SPL {X  -160.000, Y  +563.667, Z    +0.000, E1   -45.146, E3 +92654.542}
SPL {X  -160.000, Y  +574.965, Z    +0.000, E1   -45.125, E3 +92678.518}
SPL {X  -160.000, Y  +585.644, Z    +0.000, E1   -45.117, E3 +92701.158}
SPL {X  -160.000, Y  +596.819, Z    +0.000, E1   -45.144, E3 +92724.799}
SPL {X  -160.000, Y  +608.165, Z    +0.000, E1   -45.120, E3 +92748.874}
SPL {X  -160.000, Y  +619.270, Z    +0.000, E1   -45.132, E3 +92772.376}
SPL {X  -160.000, Y  +629.968, Z    +0.000, E1   -45.117, E3 +92795.042}
SPL {X  -160.000, Y  +640.750, Z    +0.000, E1   -45.131, E3 +92817.865}
SPL {X  -160.000, Y  +651.429, Z    +0.000, E1   -45.117, E3 +92840.507}
SPL {X  -160.000, Y  +662.434, Z    +0.000, E1   -45.129, E3 +92863.851}
SPL {X  -159.992, Y  +673.110, Z    +0.000, E1   -45.097, E3 +92886.543}
SPL {X  -159.521, Y  +683.874, Z    +0.000, E1   -45.054, E3 +92909.799}
SPL {X  -158.435, Y  +693.823, Z    +0.000, E1   -44.810, E3 +92932.103}
SPL {X  -156.807, Y  +703.304, Z    +0.000, E1   -44.558, E3 +92953.823}
SPL {X  -154.802, Y  +711.950, Z    +0.000, E1   -44.141, E3 +92974.283}
SPL {X  -152.641, Y  +719.464, Z    +0.000, E1   -43.749, E3 +92992.399}
SPL {X  -149.826, Y  +727.645, Z    +0.000, E1   -43.252, E3 +93012.502}
SPL {X  -145.307, Y  +738.478, Z    +0.000, E1   -36.676, E3 +93092.570}
ENDSPLINE

SPLINE
SPL {X  -155.601, Y  +708.762, Z    +0.000, E1   -21.463, E3 +93147.356}
SPL {X  -158.549, Y  +693.002, Z    +0.000, E1   -13.406, E3 +93156.347}
SPL {X  -159.716, Y  +681.031, Z    +0.000, E1    -6.529, E3 +93160.497}
SPL {X  -160.000, Y  +671.641, Z    +0.000, E1    -0.547, E3 +93162.214}
SPL {X  -160.000, Y  +665.424, Z    +0.000, E1    +5.044, E3 +93163.162}
SPL {X  -160.000, Y  +658.015, Z    +0.000, E1   +12.630, E3 +93165.080}
SPL {X  -160.000, Y  +645.110, Z    +0.000, E1   +25.142, E3 +93170.880}
SPL {X  -160.000, Y  +611.664, Z    +0.000, E1   +41.262, E3 +93200.609}
SPL {X  -160.000, Y  +581.433, Z    +0.000, E1   +44.103, E3 +93250.346}
SPL {X  -160.000, Y  +572.090, Z    +0.000, E1   +44.120, E3 +93270.811}
SPL {X  -160.000, Y  +563.431, Z    +0.000, E1   +44.084, E3 +93289.864}
SPL {X  -160.000, Y  +556.107, Z    +0.000, E1   +44.076, E3 +93305.932}
SPL {X  -160.000, Y  +549.181, Z    +0.000, E1   +44.079, E3 +93321.092}
SPL {X  -160.000, Y  +542.413, Z    +0.000, E1   +44.088, E3 +93335.926}
SPL {X  -160.000, Y  +534.609, Z    +0.000, E1   +44.095, E3 +93353.036}
SPL {X  -160.000, Y  +527.457, Z    +0.000, E1   +44.070, E3 +93368.746}
SPL {X  -160.000, Y  +520.912, Z    +0.000, E1   +44.079, E3 +93383.087}
SPL {X  -160.000, Y  +514.086, Z    +0.000, E1   +44.081, E3 +93398.035}
SPL {X  -160.000, Y  +507.208, Z    +0.000, E1   +44.082, E3 +93413.112}
SPL {X  -160.000, Y  +499.184, Z    +0.000, E1   +44.113, E3 +93430.670}
ENDSPLINE

SPLINE
SPL {X  -160.000, Y  +503.824, Z    +0.000, E1   +39.488, E3 +93446.718}
ENDSPLINE

SPLINE
SPL {X  -160.000, Y  +499.279, Z    +0.000, E1   +38.981, E3 +93461.708}
SPL {X  -160.000, Y  +490.068, Z    +0.000, E1   +40.198, E3 +93478.013}
SPL {X  -160.000, Y  +481.368, Z    +0.000, E1   +41.274, E3 +93493.002}
SPL {X  -160.000, Y  +470.910, Z    +0.000, E1   +42.658, E3 +93509.511}
SPL {X  -160.000, Y  +460.219, Z    +0.000, E1   +43.912, E3 +93526.132}
SPL {X  -160.000, Y  +451.951, Z    +0.000, E1   +44.355, E3 +93541.697}
SPL {X  -160.000, Y  +442.331, Z    +0.000, E1   +44.390, E3 +93562.561}
SPL {X  -160.000, Y  +433.037, Z    +0.000, E1   +44.348, E3 +93582.835}
SPL {X  -160.000, Y  +424.435, Z    +0.000, E1   +44.358, E3 +93601.504}
SPL {X  -160.000, Y  +416.015, Z    +0.000, E1   +44.348, E3 +93619.824}
SPL {X  -160.000, Y  +407.167, Z    +0.000, E1   +44.365, E3 +93639.035}
SPL {X  -160.000, Y  +397.599, Z    +0.000, E1   +44.371, E3 +93659.843}
SPL {X  -160.000, Y  +388.533, Z    +0.000, E1   +44.340, E3 +93679.618}
SPL {X  -159.759, Y  +380.021, Z    +0.000, E1   +44.311, E3 +93698.350}
SPL {X  -159.014, Y  +371.065, Z    +0.000, E1   +44.193, E3 +93718.588}
SPL {X  -157.745, Y  +362.030, Z    +0.000, E1   +43.965, E3 +93739.570}
SPL {X  -156.258, Y  +354.400, Z    +0.000, E1   +43.653, E3 +93757.777}
SPL {X  -154.385, Y  +346.786, Z    +0.000, E1   +43.356, E3 +93776.189}
SPL {X  -152.146, Y  +339.286, Z    +0.000, E1   +42.904, E3 +93794.824}
SPL {X  -149.854, Y  +332.731, Z    +0.000, E1   +42.474, E3 +93811.351}
SPL {X  -145.635, Y  +322.541, Z    +0.000, E1   +36.397, E3 +93887.310}
ENDSPLINE

SPLINE
SPL {X  -156.682, Y  +356.385, Z    +0.000, E1   +19.033, E3 +93945.616}
SPL {X  -159.526, Y  +376.492, Z    +0.000, E1    +8.067, E3 +93955.525}
SPL {X  -159.961, Y  +385.275, Z    +0.000, E1    +2.550, E3 +93957.564}
SPL {X  -160.000, Y  +390.345, Z    +0.000, E1    -1.188, E3 +93958.290}
SPL {X  -160.000, Y  +395.838, Z    +0.000, E1    -6.211, E3 +93959.233}
SPL {X  -160.000, Y  +403.277, Z    +0.000, E1   -14.057, E3 +93961.185}
SPL {X  -160.000, Y  +414.316, Z    +0.000, E1   -24.810, E3 +93966.258}
SPL {X  -160.000, Y  +442.604, Z    +0.000, E1   -40.161, E3 +93988.392}
SPL {X  -160.000, Y  +482.867, Z    +0.000, E1   -45.148, E3 +94048.608}
SPL {X  -160.000, Y  +494.769, Z    +0.000, E1   -45.151, E3 +94073.827}
SPL {X  -160.000, Y  +505.761, Z    +0.000, E1   -45.118, E3 +94097.141}
SPL {X  -160.000, Y  +517.347, Z    +0.000, E1   -45.173, E3 +94121.579}
SPL {X  -160.000, Y  +529.298, Z    +0.000, E1   -45.138, E3 +94146.962}
SPL {X  -160.000, Y  +540.664, Z    +0.000, E1   -45.139, E3 +94171.040}
SPL {X  -160.000, Y  +552.011, Z    +0.000, E1   -45.139, E3 +94195.076}
SPL {X  -160.000, Y  +563.667, Z    +0.000, E1   -45.146, E3 +94219.756}
SPL {X  -160.000, Y  +574.965, Z    +0.000, E1   -45.125, E3 +94243.732}
SPL {X  -160.000, Y  +585.644, Z    +0.000, E1   -45.117, E3 +94266.372}
SPL {X  -160.000, Y  +596.819, Z    +0.000, E1   -45.144, E3 +94290.013}
SPL {X  -160.000, Y  +608.165, Z    +0.000, E1   -45.120, E3 +94314.088}
SPL {X  -160.000, Y  +619.270, Z    +0.000, E1   -45.132, E3 +94337.590}
SPL {X  -160.000, Y  +629.968, Z    +0.000, E1   -45.117, E3 +94360.257}
SPL {X  -160.000, Y  +640.750, Z    +0.000, E1   -45.131, E3 +94383.080}
SPL {X  -160.000, Y  +651.429, Z    +0.000, E1   -45.117, E3 +94405.721}
SPL {X  -160.000, Y  +662.434, Z    +0.000, E1   -45.129, E3 +94429.065}
SPL {X  -159.992, Y  +673.110, Z    +0.000, E1   -45.097, E3 +94451.758}
SPL {X  -159.521, Y  +683.874, Z    +0.000, E1   -45.054, E3 +94475.013}
SPL {X  -158.435, Y  +693.823, Z    +0.000, E1   -44.810, E3 +94497.317}
SPL {X  -156.807, Y  +703.304, Z    +0.000, E1   -44.558, E3 +94519.038}
SPL {X  -154.802, Y  +711.950, Z    +0.000, E1   -44.141, E3 +94539.498}
SPL {X  -152.641, Y  +719.464, Z    +0.000, E1   -43.749, E3 +94557.613}
SPL {X  -149.826, Y  +727.645, Z    +0.000, E1   -43.252, E3 +94577.716}
SPL {X  -145.307, Y  +738.478, Z    +0.000, E1   -36.676, E3 +94657.784}
ENDSPLINE

SPLINE
SPL {X  -155.601, Y  +708.762, Z    +0.000, E1   -21.463, E3 +94712.571}
SPL {X  -158.549, Y  +693.002, Z    +0.000, E1   -13.406, E3 +94721.561}
SPL {X  -159.716, Y  +681.031, Z    +0.000, E1    -6.529, E3 +94725.711}
SPL {X  -160.000, Y  +671.641, Z    +0.000, E1    -0.547, E3 +94727.428}
SPL {X  -160.000, Y  +665.424, Z    +0.000, E1    +5.044, E3 +94728.376}
SPL {X  -160.000, Y  +658.015, Z    +0.000, E1   +12.630, E3 +94730.294}
SPL {X  -160.000, Y  +645.110, Z    +0.000, E1   +25.142, E3 +94736.094}
SPL {X  -160.000, Y  +611.664, Z    +0.000, E1   +41.262, E3 +94765.824}
SPL {X  -160.000, Y  +581.433, Z    +0.000, E1   +44.103, E3 +94815.560}
SPL {X  -160.000, Y  +572.090, Z    +0.000, E1   +44.120, E3 +94836.025}
SPL {X  -160.000, Y  +563.431, Z    +0.000, E1   +44.084, E3 +94855.078}
SPL {X  -160.000, Y  +556.107, Z    +0.000, E1   +44.076, E3 +94871.146}
SPL {X  -160.000, Y  +549.181, Z    +0.000, E1   +44.079, E3 +94886.306}
SPL {X  -160.000, Y  +542.413, Z    +0.000, E1   +44.088, E3 +94901.140}
SPL {X  -160.000, Y  +534.609, Z    +0.000, E1   +44.095, E3 +94918.250}
SPL {X  -160.000, Y  +527.457, Z    +0.000, E1   +44.070, E3 +94933.960}
SPL {X  -160.000, Y  +520.912, Z    +0.000, E1   +44.079, E3 +94948.301}
SPL {X  -160.000, Y  +514.086, Z    +0.000, E1   +44.081, E3 +94963.249}
SPL {X  -160.000, Y  +507.208, Z    +0.000, E1   +44.082, E3 +94978.326}
SPL {X  -160.000, Y  +499.184, Z    +0.000, E1   +44.113, E3 +94995.884}
ENDSPLINE

SPLINE
SPL {X  -160.000, Y  +503.824, Z    +0.000, E1   +39.488, E3 +95011.933}
ENDSPLINE

SPLINE
SPL {X  -160.000, Y  +499.279, Z    +0.000, E1   +38.981, E3 +95026.923}
SPL {X  -160.000, Y  +490.068, Z    +0.000, E1   +40.198, E3 +95043.227}
SPL {X  -160.000, Y  +481.368, Z    +0.000, E1   +41.274, E3 +95058.217}
SPL {X  -160.000, Y  +470.910, Z    +0.000, E1   +42.658, E3 +95074.725}
SPL {X  -160.000, Y  +460.219, Z    +0.000, E1   +43.912, E3 +95091.346}
SPL {X  -160.000, Y  +451.951, Z    +0.000, E1   +44.355, E3 +95106.911}
SPL {X  -160.000, Y  +442.331, Z    +0.000, E1   +44.390, E3 +95127.775}
SPL {X  -160.000, Y  +433.037, Z    +0.000, E1   +44.348, E3 +95148.050}
SPL {X  -160.000, Y  +424.435, Z    +0.000, E1   +44.358, E3 +95166.718}
SPL {X  -160.000, Y  +416.015, Z    +0.000, E1   +44.348, E3 +95185.038}
SPL {X  -160.000, Y  +407.167, Z    +0.000, E1   +44.365, E3 +95204.249}
SPL {X  -160.000, Y  +397.599, Z    +0.000, E1   +44.371, E3 +95225.057}
SPL {X  -160.000, Y  +388.533, Z    +0.000, E1   +44.340, E3 +95244.832}
SPL {X  -159.759, Y  +380.021, Z    +0.000, E1   +44.311, E3 +95263.564}
SPL {X  -159.014, Y  +371.065, Z    +0.000, E1   +44.193, E3 +95283.802}
SPL {X  -157.745, Y  +362.030, Z    +0.000, E1   +43.965, E3 +95304.784}
SPL {X  -156.258, Y  +354.400, Z    +0.000, E1   +43.653, E3 +95322.991}
SPL {X  -154.385, Y  +346.786, Z    +0.000, E1   +43.356, E3 +95341.403}
SPL {X  -152.146, Y  +339.286, Z    +0.000, E1   +42.904, E3 +95360.038}
SPL {X  -149.854, Y  +332.731, Z    +0.000, E1   +42.474, E3 +95376.565}
SPL {X  -145.635, Y  +322.541, Z    +0.000, E1   +36.397, E3 +95452.524}
ENDSPLINE

SPLINE
SPL {X  -156.682, Y  +356.385, Z    +0.000, E1   +19.033, E3 +95510.831}
SPL {X  -159.526, Y  +376.492, Z    +0.000, E1    +8.067, E3 +95520.740}
SPL {X  -159.961, Y  +385.275, Z    +0.000, E1    +2.550, E3 +95522.778}
SPL {X  -160.000, Y  +390.345, Z    +0.000, E1    -1.188, E3 +95523.504}
SPL {X  -160.000, Y  +395.838, Z    +0.000, E1    -6.211, E3 +95524.448}
SPL {X  -160.000, Y  +403.277, Z    +0.000, E1   -14.057, E3 +95526.399}
SPL {X  -160.000, Y  +414.316, Z    +0.000, E1   -24.810, E3 +95531.472}
SPL {X  -160.000, Y  +442.604, Z    +0.000, E1   -40.161, E3 +95553.606}
SPL {X  -160.000, Y  +482.867, Z    +0.000, E1   -45.148, E3 +95613.822}
SPL {X  -160.000, Y  +494.769, Z    +0.000, E1   -45.151, E3 +95639.041}
SPL {X  -160.000, Y  +505.761, Z    +0.000, E1   -45.118, E3 +95662.355}
SPL {X  -160.000, Y  +517.347, Z    +0.000, E1   -45.173, E3 +95686.793}
SPL {X  -160.000, Y  +529.298, Z    +0.000, E1   -45.138, E3 +95712.176}
SPL {X  -160.000, Y  +540.664, Z    +0.000, E1   -45.139, E3 +95736.254}
SPL {X  -160.000, Y  +552.011, Z    +0.000, E1   -45.139, E3 +95760.290}
SPL {X  -160.000, Y  +563.667, Z    +0.000, E1   -45.146, E3 +95784.970}
SPL {X  -160.000, Y  +574.965, Z    +0.000, E1   -45.125, E3 +95808.946}
SPL {X  -160.000, Y  +585.644, Z    +0.000, E1   -45.117, E3 +95831.586}
SPL {X  -160.000, Y  +596.819, Z    +0.000, E1   -45.144, E3 +95855.228}
SPL {X  -160.000, Y  +608.165, Z    +0.000, E1   -45.120, E3 +95879.302}
SPL {X  -160.000, Y  +619.270, Z    +0.000, E1   -45.132, E3 +95902.805}
SPL {X  -160.000, Y  +629.968, Z    +0.000, E1   -45.117, E3 +95925.471}
SPL {X  -160.000, Y  +640.750, Z    +0.000, E1   -45.131, E3 +95948.294}
SPL {X  -160.000, Y  +651.429, Z    +0.000, E1   -45.117, E3 +95970.935}
SPL {X  -160.000, Y  +662.434, Z    +0.000, E1   -45.129, E3 +95994.279}
SPL {X  -159.992, Y  +673.110, Z    +0.000, E1   -45.097, E3 +96016.972}
SPL {X  -159.521, Y  +683.874, Z    +0.000, E1   -45.054, E3 +96040.227}
SPL {X  -158.435, Y  +693.823, Z    +0.000, E1   -44.810, E3 +96062.531}
SPL {X  -156.807, Y  +703.304, Z    +0.000, E1   -44.558, E3 +96084.252}
SPL {X  -154.802, Y  +711.950, Z    +0.000, E1   -44.141, E3 +96104.712}
SPL {X  -152.641, Y  +719.464, Z    +0.000, E1   -43.749, E3 +96122.828}
SPL {X  -149.826, Y  +727.645, Z    +0.000, E1   -43.252, E3 +96142.930}
SPL {X  -145.307, Y  +738.478, Z    +0.000, E1   -36.676, E3 +96222.998}
ENDSPLINE

SPLINE
SPL {X  -155.601, Y  +708.762, Z    +0.000, E1   -21.463, E3 +96277.785}
SPL {X  -158.549, Y  +693.002, Z    +0.000, E1   -13.406, E3 +96286.776}
SPL {X  -159.716, Y  +681.031, Z    +0.000, E1    -6.529, E3 +96290.926}
SPL {X  -160.000, Y  +671.641, Z    +0.000, E1    -0.547, E3 +96292.642}
SPL {X  -160.000, Y  +665.424, Z    +0.000, E1    +5.044, E3 +96293.590}
SPL {X  -160.000, Y  +658.015, Z    +0.000, E1   +12.630, E3 +96295.508}
SPL {X  -160.000, Y  +645.110, Z    +0.000, E1   +25.142, E3 +96301.308}
SPL {X  -160.000, Y  +611.664, Z    +0.000, E1   +41.262, E3 +96331.038}
SPL {X  -160.000, Y  +581.433, Z    +0.000, E1   +44.103, E3 +96380.774}
SPL {X  -160.000, Y  +572.090, Z    +0.000, E1   +44.120, E3 +96401.239}
SPL {X  -160.000, Y  +563.431, Z    +0.000, E1   +44.084, E3 +96420.292}
SPL {X  -160.000, Y  +556.107, Z    +0.000, E1   +44.076, E3 +96436.360}
SPL {X  -160.000, Y  +549.181, Z    +0.000, E1   +44.079, E3 +96451.520}
SPL {X  -160.000, Y  +542.413, Z    +0.000, E1   +44.088, E3 +96466.354}
SPL {X  -160.000, Y  +534.609, Z    +0.000, E1   +44.095, E3 +96483.464}
SPL {X  -160.000, Y  +527.457, Z    +0.000, E1   +44.070, E3 +96499.174}
SPL {X  -160.000, Y  +520.912, Z    +0.000, E1   +44.079, E3 +96513.515}
SPL {X  -160.000, Y  +514.086, Z    +0.000, E1   +44.081, E3 +96528.464}
SPL {X  -160.000, Y  +507.208, Z    +0.000, E1   +44.082, E3 +96543.540}
SPL {X  -160.000, Y  +499.184, Z    +0.000, E1   +44.113, E3 +96561.098}
ENDSPLINE

SPLINE
SPL {X  -160.000, Y  +503.824, Z    +0.000, E1   +39.488, E3 +96577.147}
ENDSPLINE

SPLINE
SPL {X  -160.000, Y  +499.279, Z    +0.000, E1   +38.981, E3 +96592.137}
SPL {X  -160.000, Y  +490.068, Z    +0.000, E1   +40.198, E3 +96608.441}
SPL {X  -160.000, Y  +481.368, Z    +0.000, E1   +41.274, E3 +96623.431}
SPL {X  -160.000, Y  +470.910, Z    +0.000, E1   +42.658, E3 +96639.939}
SPL {X  -160.000, Y  +460.219, Z    +0.000, E1   +43.912, E3 +96656.560}
SPL {X  -160.000, Y  +451.951, Z    +0.000, E1   +44.355, E3 +96672.126}
SPL {X  -160.000, Y  +442.331, Z    +0.000, E1   +44.390, E3 +96692.990}
SPL {X  -160.000, Y  +433.037, Z    +0.000, E1   +44.348, E3 +96713.264}
SPL {X  -160.000, Y  +424.435, Z    +0.000, E1   +44.358, E3 +96731.932}
SPL {X  -160.000, Y  +416.015, Z    +0.000, E1   +44.348, E3 +96750.252}
SPL {X  -160.000, Y  +407.167, Z    +0.000, E1   +44.365, E3 +96769.463}
SPL {X  -160.000, Y  +397.599, Z    +0.000, E1   +44.371, E3 +96790.271}
SPL {X  -160.000, Y  +388.533, Z    +0.000, E1   +44.340, E3 +96810.046}
SPL {X  -159.759, Y  +380.021, Z    +0.000, E1   +44.311, E3 +96828.778}
SPL {X  -159.014, Y  +371.065, Z    +0.000, E1   +44.193, E3 +96849.016}
SPL {X  -157.745, Y  +362.030, Z    +0.000, E1   +43.965, E3 +96869.998}
SPL {X  -156.258, Y  +354.400, Z    +0.000, E1   +43.653, E3 +96888.206}
SPL {X  -154.385, Y  +346.786, Z    +0.000, E1   +43.356, E3 +96906.617}
SPL {X  -152.146, Y  +339.286, Z    +0.000, E1   +42.904, E3 +96925.252}
SPL {X  -149.854, Y  +332.731, Z    +0.000, E1   +42.474, E3 +96941.780}
SPL {X  -145.635, Y  +322.541, Z    +0.000, E1   +36.397, E3 +97017.739}
ENDSPLINE

SPLINE
SPL {X  -156.682, Y  +356.385, Z    +0.000, E1   +19.033, E3 +97076.045}
SPL {X  -159.526, Y  +376.492, Z    +0.000, E1    +8.067, E3 +97085.954}
SPL {X  -159.961, Y  +385.275, Z    +0.000, E1    +2.550, E3 +97087.992}
SPL {X  -160.000, Y  +390.345, Z    +0.000, E1    -1.188, E3 +97088.718}
SPL {X  -160.000, Y  +395.838, Z    +0.000, E1    -6.211, E3 +97089.662}
SPL {X  -160.000, Y  +403.277, Z    +0.000, E1   -14.057, E3 +97091.613}
SPL {X  -160.000, Y  +414.316, Z    +0.000, E1   -24.810, E3 +97096.686}
SPL {X  -160.000, Y  +442.604, Z    +0.000, E1   -40.161, E3 +97118.820}
SPL {X  -160.000, Y  +482.867, Z    +0.000, E1   -45.148, E3 +97179.036}
SPL {X  -160.000, Y  +494.769, Z    +0.000, E1   -45.151, E3 +97204.255}
SPL {X  -160.000, Y  +505.761, Z    +0.000, E1   -45.118, E3 +97227.569}
SPL {X  -160.000, Y  +517.347, Z    +0.000, E1   -45.173, E3 +97252.007}
SPL {X  -160.000, Y  +529.298, Z    +0.000, E1   -45.138, E3 +97277.390}
SPL {X  -160.000, Y  +540.664, Z    +0.000, E1   -45.139, E3 +97301.468}
SPL {X  -160.000, Y  +552.011, Z    +0.000, E1   -45.139, E3 +97325.504}
SPL {X  -160.000, Y  +563.667, Z    +0.000, E1   -45.146, E3 +97350.185}
SPL {X  -160.000, Y  +574.965, Z    +0.000, E1   -45.125, E3 +97374.160}
SPL {X  -160.000, Y  +585.644, Z    +0.000, E1   -45.117, E3 +97396.800}
SPL {X  -160.000, Y  +596.819, Z    +0.000, E1   -45.144, E3 +97420.442}
SPL {X  -160.000, Y  +608.165, Z    +0.000, E1   -45.120, E3 +97444.516}
SPL {X  -160.000, Y  +619.270, Z    +0.000, E1   -45.132, E3 +97468.019}
SPL {X  -160.000, Y  +629.968, Z    +0.000, E1   -45.117, E3 +97490.685}
SPL {X  -160.000, Y  +640.750, Z    +0.000, E1   -45.131, E3 +97513.508}
SPL {X  -160.000, Y  +651.429, Z    +0.000, E1   -45.117, E3 +97536.149}
SPL {X  -160.000, Y  +662.434, Z    +0.000, E1   -45.129, E3 +97559.493}
SPL {X  -159.992, Y  +673.110, Z    +0.000, E1   -45.097, E3 +97582.186}
SPL {X  -159.521, Y  +683.874, Z    +0.000, E1   -45.054, E3 +97605.441}
SPL {X  -158.435, Y  +693.823, Z    +0.000, E1   -44.810, E3 +97627.745}
SPL {X  -156.807, Y  +703.304, Z    +0.000, E1   -44.558, E3 +97649.466}
SPL {X  -154.802, Y  +711.950, Z    +0.000, E1   -44.141, E3 +97669.926}
SPL {X  -152.641, Y  +719.464, Z    +0.000, E1   -43.749, E3 +97688.042}
SPL {X  -149.826, Y  +727.645, Z    +0.000, E1   -43.252, E3 +97708.145}
SPL {X  -145.307, Y  +738.478, Z    +0.000, E1   -36.676, E3 +97788.212}
ENDSPLINE

SPLINE
SPL {X  -155.601, Y  +708.762, Z    +0.000, E1   -21.463, E3 +97842.999}
SPL {X  -158.549, Y  +693.002, Z    +0.000, E1   -13.406, E3 +97851.990}
SPL {X  -159.716, Y  +681.031, Z    +0.000, E1    -6.529, E3 +97856.140}
SPL {X  -160.000, Y  +671.641, Z    +0.000, E1    -0.547, E3 +97857.856}
SPL {X  -160.000, Y  +665.424, Z    +0.000, E1    +5.044, E3 +97858.805}
SPL {X  -160.000, Y  +658.015, Z    +0.000, E1   +12.630, E3 +97860.722}
SPL {X  -160.000, Y  +645.110, Z    +0.000, E1   +25.142, E3 +97866.523}
SPL {X  -160.000, Y  +611.664, Z    +0.000, E1   +41.262, E3 +97896.252}
SPL {X  -160.000, Y  +581.433, Z    +0.000, E1   +44.103, E3 +97945.989}
SPL {X  -160.000, Y  +572.090, Z    +0.000, E1   +44.120, E3 +97966.453}
SPL {X  -160.000, Y  +563.431, Z    +0.000, E1   +44.084, E3 +97985.506}
SPL {X  -160.000, Y  +556.107, Z    +0.000, E1   +44.076, E3 +98001.575}
SPL {X  -160.000, Y  +549.181, Z    +0.000, E1   +44.079, E3 +98016.734}
SPL {X  -160.000, Y  +542.413, Z    +0.000, E1   +44.088, E3 +98031.568}
SPL {X  -160.000, Y  +534.609, Z    +0.000, E1   +44.095, E3 +98048.678}
SPL {X  -160.000, Y  +527.457, Z    +0.000, E1   +44.070, E3 +98064.389}
SPL {X  -160.000, Y  +520.912, Z    +0.000, E1   +44.079, E3 +98078.729}
SPL {X  -160.000, Y  +514.086, Z    +0.000, E1   +44.081, E3 +98093.678}
SPL {X  -160.000, Y  +507.208, Z    +0.000, E1   +44.082, E3 +98108.754}
SPL {X  -160.000, Y  +499.184, Z    +0.000, E1   +44.113, E3 +98126.312}
ENDSPLINE

SPLINE
SPL {X  -160.000, Y  +503.824, Z    +0.000, E1   +39.488, E3 +98142.361}
ENDSPLINE

SPLINE
SPL {X  -160.000, Y  +499.279, Z    +0.000, E1   +38.981, E3 +98157.351}
SPL {X  -160.000, Y  +490.068, Z    +0.000, E1   +40.198, E3 +98173.655}
SPL {X  -160.000, Y  +481.368, Z    +0.000, E1   +41.274, E3 +98188.645}
SPL {X  -160.000, Y  +470.910, Z    +0.000, E1   +42.658, E3 +98205.154}
SPL {X  -160.000, Y  +460.219, Z    +0.000, E1   +43.912, E3 +98221.774}
SPL {X  -160.000, Y  +451.951, Z    +0.000, E1   +44.355, E3 +98237.340}
SPL {X  -160.000, Y  +442.331, Z    +0.000, E1   +44.390, E3 +98258.204}
SPL {X  -160.000, Y  +433.037, Z    +0.000, E1   +44.348, E3 +98278.478}
SPL {X  -160.000, Y  +424.435, Z    +0.000, E1   +44.358, E3 +98297.146}
SPL {X  -160.000, Y  +416.015, Z    +0.000, E1   +44.348, E3 +98315.466}
SPL {X  -160.000, Y  +407.167, Z    +0.000, E1   +44.365, E3 +98334.677}
SPL {X  -160.000, Y  +397.599, Z    +0.000, E1   +44.371, E3 +98355.485}
SPL {X  -160.000, Y  +388.533, Z    +0.000, E1   +44.340, E3 +98375.260}
SPL {X  -159.759, Y  +380.021, Z    +0.000, E1   +44.311, E3 +98393.992}
SPL {X  -159.014, Y  +371.065, Z    +0.000, E1   +44.193, E3 +98414.230}
SPL {X  -157.745, Y  +362.030, Z    +0.000, E1   +43.965, E3 +98435.212}
SPL {X  -156.258, Y  +354.400, Z    +0.000, E1   +43.653, E3 +98453.420}
SPL {X  -154.385, Y  +346.786, Z    +0.000, E1   +43.356, E3 +98471.831}
SPL {X  -152.146, Y  +339.286, Z    +0.000, E1   +42.904, E3 +98490.466}
SPL {X  -149.854, Y  +332.731, Z    +0.000, E1   +42.474, E3 +98506.994}
SPL {X  -145.635, Y  +322.541, Z    +0.000, E1   +36.397, E3 +98582.953}
ENDSPLINE

SPLINE
SPL {X  -156.682, Y  +356.385, Z    +0.000, E1   +19.033, E3 +98641.259}
SPL {X  -159.526, Y  +376.492, Z    +0.000, E1    +8.067, E3 +98651.168}
SPL {X  -159.961, Y  +385.275, Z    +0.000, E1    +2.550, E3 +98653.206}
SPL {X  -160.000, Y  +390.345, Z    +0.000, E1    -1.188, E3 +98653.932}
SPL {X  -160.000, Y  +395.838, Z    +0.000, E1    -6.211, E3 +98654.876}
SPL {X  -160.000, Y  +403.277, Z    +0.000, E1   -14.057, E3 +98656.827}
SPL {X  -160.000, Y  +414.316, Z    +0.000, E1   -24.810, E3 +98661.900}
SPL {X  -160.000, Y  +442.604, Z    +0.000, E1   -40.161, E3 +98684.034}
SPL {X  -160.000, Y  +482.867, Z    +0.000, E1   -45.148, E3 +98744.250}
SPL {X  -160.000, Y  +494.769, Z    +0.000, E1   -45.151, E3 +98769.470}
SPL {X  -160.000, Y  +505.761, Z    +0.000, E1   -45.118, E3 +98792.784}
SPL {X  -160.000, Y  +517.347, Z    +0.000, E1   -45.173, E3 +98817.221}
SPL {X  -160.000, Y  +529.298, Z    +0.000, E1   -45.138, E3 +98842.605}
SPL {X  -160.000, Y  +540.664, Z    +0.000, E1   -45.139, E3 +98866.682}
SPL {X  -160.000, Y  +552.011, Z    +0.000, E1   -45.139, E3 +98890.718}
SPL {X  -160.000, Y  +563.667, Z    +0.000, E1   -45.146, E3 +98915.399}
SPL {X  -160.000, Y  +574.965, Z    +0.000, E1   -45.125, E3 +98939.374}
SPL {X  -160.000, Y  +585.644, Z    +0.000, E1   -45.117, E3 +98962.014}
SPL {X  -160.000, Y  +596.819, Z    +0.000, E1   -45.144, E3 +98985.656}
SPL {X  -160.000, Y  +608.165, Z    +0.000, E1   -45.120, E3 +99009.730}
SPL {X  -160.000, Y  +619.270, Z    +0.000, E1   -45.132, E3 +99033.233}
SPL {X  -160.000, Y  +629.968, Z    +0.000, E1   -45.117, E3 +99055.899}
SPL {X  -160.000, Y  +640.750, Z    +0.000, E1   -45.131, E3 +99078.722}
SPL {X  -160.000, Y  +651.429, Z    +0.000, E1   -45.117, E3 +99101.363}
SPL {X  -160.000, Y  +662.434, Z    +0.000, E1   -45.129, E3 +99124.707}
SPL {X  -159.992, Y  +673.110, Z    +0.000, E1   -45.097, E3 +99147.400}
SPL {X  -159.521, Y  +683.874, Z    +0.000, E1   -45.054, E3 +99170.655}
SPL {X  -158.435, Y  +693.823, Z    +0.000, E1   -44.810, E3 +99192.959}
SPL {X  -156.807, Y  +703.304, Z    +0.000, E1   -44.558, E3 +99214.680}
SPL {X  -154.802, Y  +711.950, Z    +0.000, E1   -44.141, E3 +99235.140}
SPL {X  -152.641, Y  +719.464, Z    +0.000, E1   -43.749, E3 +99253.256}
SPL {X  -149.826, Y  +727.645, Z    +0.000, E1   -43.252, E3 +99273.359}
SPL {X  -145.307, Y  +738.478, Z    +0.000, E1   -36.676, E3 +99353.426}
ENDSPLINE

SPLINE
SPL {X  -155.601, Y  +708.762, Z    +0.000, E1   -21.463, E3 +99408.213}
SPL {X  -158.549, Y  +693.002, Z    +0.000, E1   -13.406, E3 +99417.204}
SPL {X  -159.716, Y  +681.031, Z    +0.000, E1    -6.529, E3 +99421.354}
SPL {X  -160.000, Y  +671.641, Z    +0.000, E1    -0.547, E3 +99423.071}
SPL {X  -160.000, Y  +665.424, Z    +0.000, E1    +5.044, E3 +99424.019}
SPL {X  -160.000, Y  +658.015, Z    +0.000, E1   +12.630, E3 +99425.937}
SPL {X  -160.000, Y  +645.110, Z    +0.000, E1   +25.142, E3 +99431.737}
SPL {X  -160.000, Y  +611.664, Z    +0.000, E1   +41.262, E3 +99461.466}
SPL {X  -160.000, Y  +581.433, Z    +0.000, E1   +44.103, E3 +99511.203}
SPL {X  -160.000, Y  +572.090, Z    +0.000, E1   +44.120, E3 +99531.667}
SPL {X  -160.000, Y  +563.431, Z    +0.000, E1   +44.084, E3 +99550.720}
SPL {X  -160.000, Y  +556.107, Z    +0.000, E1   +44.076, E3 +99566.789}
SPL {X  -160.000, Y  +549.181, Z    +0.000, E1   +44.079, E3 +99581.948}
SPL {X  -160.000, Y  +542.413, Z    +0.000, E1   +44.088, E3 +99596.782}
SPL {X  -160.000, Y  +534.609, Z    +0.000, E1   +44.095, E3 +99613.892}
SPL {X  -160.000, Y  +527.457, Z    +0.000, E1   +44.070, E3 +99629.603}
SPL {X  -160.000, Y  +520.912, Z    +0.000, E1   +44.079, E3 +99643.944}
SPL {X  -160.000, Y  +514.086, Z    +0.000, E1   +44.081, E3 +99658.892}
SPL {X  -160.000, Y  +507.208, Z    +0.000, E1   +44.082, E3 +99673.968}
SPL {X  -160.000, Y  +499.184, Z    +0.000, E1   +44.113, E3 +99691.526}
ENDSPLINE

SPLINE
SPL {X  -160.000, Y  +503.824, Z    +0.000, E1   +39.488, E3 +99707.575}
ENDSPLINE

SPLINE
SPL {X  -160.000, Y  +499.279, Z    +0.000, E1   +38.981, E3 +99722.565}
SPL {X  -160.000, Y  +490.068, Z    +0.000, E1   +40.198, E3 +99738.869}
SPL {X  -160.000, Y  +481.368, Z    +0.000, E1   +41.274, E3 +99753.859}
SPL {X  -160.000, Y  +470.910, Z    +0.000, E1   +42.658, E3 +99770.368}
SPL {X  -160.000, Y  +460.219, Z    +0.000, E1   +43.912, E3 +99786.988}
SPL {X  -160.000, Y  +451.951, Z    +0.000, E1   +44.355, E3 +99802.554}
SPL {X  -160.000, Y  +442.331, Z    +0.000, E1   +44.390, E3 +99823.418}
SPL {X  -160.000, Y  +433.037, Z    +0.000, E1   +44.348, E3 +99843.692}
SPL {X  -160.000, Y  +424.435, Z    +0.000, E1   +44.358, E3 +99862.360}
SPL {X  -160.000, Y  +416.015, Z    +0.000, E1   +44.348, E3 +99880.680}
SPL {X  -160.000, Y  +407.167, Z    +0.000, E1   +44.365, E3 +99899.891}
SPL {X  -160.000, Y  +397.599, Z    +0.000, E1   +44.371, E3 +99920.699}
SPL {X  -160.000, Y  +388.533, Z    +0.000, E1   +44.340, E3 +99940.474}
SPL {X  -159.759, Y  +380.021, Z    +0.000, E1   +44.311, E3 +99959.206}
SPL {X  -159.014, Y  +371.065, Z    +0.000, E1   +44.193, E3 +99979.444}
SPL {X  -157.745, Y  +362.030, Z    +0.000, E1   +43.965, E3 +100000.426}
SPL {X  -156.258, Y  +354.400, Z    +0.000, E1   +43.653, E3 +100018.634}
SPL {X  -154.385, Y  +346.786, Z    +0.000, E1   +43.356, E3 +100037.046}
SPL {X  -152.146, Y  +339.286, Z    +0.000, E1   +42.904, E3 +100055.680}
SPL {X  -149.854, Y  +332.731, Z    +0.000, E1   +42.474, E3 +100072.208}
SPL {X  -145.635, Y  +322.541, Z    +0.000, E1   +36.397, E3 +100148.167}
ENDSPLINE

SPLINE
SPL {X  -156.682, Y  +356.385, Z    +0.000, E1   +19.033, E3 +100206.473}
SPL {X  -159.526, Y  +376.492, Z    +0.000, E1    +8.067, E3 +100216.382}
SPL {X  -159.961, Y  +385.275, Z    +0.000, E1    +2.550, E3 +100218.421}
SPL {X  -160.000, Y  +390.345, Z    +0.000, E1    -1.188, E3 +100219.147}
SPL {X  -160.000, Y  +395.838, Z    +0.000, E1    -6.211, E3 +100220.090}
SPL {X  -160.000, Y  +403.277, Z    +0.000, E1   -14.057, E3 +100222.041}
SPL {X  -160.000, Y  +414.316, Z    +0.000, E1   -24.810, E3 +100227.114}
SPL {X  -160.000, Y  +442.604, Z    +0.000, E1   -40.161, E3 +100249.248}
SPL {X  -160.000, Y  +482.867, Z    +0.000, E1   -45.148, E3 +100309.464}
SPL {X  -160.000, Y  +494.769, Z    +0.000, E1   -45.151, E3 +100334.684}
SPL {X  -160.000, Y  +505.761, Z    +0.000, E1   -45.118, E3 +100357.998}
SPL {X  -160.000, Y  +517.347, Z    +0.000, E1   -45.173, E3 +100382.435}
SPL {X  -160.000, Y  +529.298, Z    +0.000, E1   -45.138, E3 +100407.819}
SPL {X  -160.000, Y  +540.664, Z    +0.000, E1   -45.139, E3 +100431.897}
SPL {X  -160.000, Y  +552.011, Z    +0.000, E1   -45.139, E3 +100455.932}
SPL {X  -160.000, Y  +563.667, Z    +0.000, E1   -45.146, E3 +100480.613}
SPL {X  -160.000, Y  +574.965, Z    +0.000, E1   -45.125, E3 +100504.588}
SPL {X  -160.000, Y  +585.644, Z    +0.000, E1   -45.117, E3 +100527.228}
SPL {X  -160.000, Y  +596.819, Z    +0.000, E1   -45.144, E3 +100550.870}
SPL {X  -160.000, Y  +608.165, Z    +0.000, E1   -45.120, E3 +100574.944}
SPL {X  -160.000, Y  +619.270, Z    +0.000, E1   -45.132, E3 +100598.447}
SPL {X  -160.000, Y  +629.968, Z    +0.000, E1   -45.117, E3 +100621.113}
SPL {X  -160.000, Y  +640.750, Z    +0.000, E1   -45.131, E3 +100643.936}
SPL {X  -160.000, Y  +651.429, Z    +0.000, E1   -45.117, E3 +100666.578}
SPL {X  -160.000, Y  +662.434, Z    +0.000, E1   -45.129, E3 +100689.921}
SPL {X  -159.992, Y  +673.110, Z    +0.000, E1   -45.097, E3 +100712.614}
SPL {X  -159.521, Y  +683.874, Z    +0.000, E1   -45.054, E3 +100735.869}
SPL {X  -158.435, Y  +693.823, Z    +0.000, E1   -44.810, E3 +100758.174}
SPL {X  -156.807, Y  +703.304, Z    +0.000, E1   -44.558, E3 +100779.894}
SPL {X  -154.802, Y  +711.950, Z    +0.000, E1   -44.141, E3 +100800.354}
SPL {X  -152.641, Y  +719.464, Z    +0.000, E1   -43.749, E3 +100818.470}
SPL {X  -149.826, Y  +727.645, Z    +0.000, E1   -43.252, E3 +100838.573}
SPL {X  -145.307, Y  +738.478, Z    +0.000, E1   -36.676, E3 +100918.640}
ENDSPLINE

SPLINE
SPL {X  -155.601, Y  +708.762, Z    +0.000, E1   -21.463, E3 +100973.427}
SPL {X  -158.549, Y  +693.002, Z    +0.000, E1   -13.406, E3 +100982.418}
SPL {X  -159.716, Y  +681.031, Z    +0.000, E1    -6.529, E3 +100986.568}
SPL {X  -160.000, Y  +671.641, Z    +0.000, E1    -0.547, E3 +100988.285}
SPL {X  -160.000, Y  +665.424, Z    +0.000, E1    +5.044, E3 +100989.233}
SPL {X  -160.000, Y  +658.015, Z    +0.000, E1   +12.630, E3 +100991.151}
SPL {X  -160.000, Y  +645.110, Z    +0.000, E1   +25.142, E3 +100996.951}
SPL {X  -160.000, Y  +611.664, Z    +0.000, E1   +41.262, E3 +101026.680}
SPL {X  -160.000, Y  +581.433, Z    +0.000, E1   +44.103, E3 +101076.417}
SPL {X  -160.000, Y  +572.090, Z    +0.000, E1   +44.120, E3 +101096.881}
SPL {X  -160.000, Y  +563.431, Z    +0.000, E1   +44.084, E3 +101115.935}
SPL {X  -160.000, Y  +556.107, Z    +0.000, E1   +44.076, E3 +101132.003}
SPL {X  -160.000, Y  +549.181, Z    +0.000, E1   +44.079, E3 +101147.162}
SPL {X  -160.000, Y  +542.413, Z    +0.000, E1   +44.088, E3 +101161.996}
SPL {X  -160.000, Y  +534.609, Z    +0.000, E1   +44.095, E3 +101179.106}
SPL {X  -160.000, Y  +527.457, Z    +0.000, E1   +44.070, E3 +101194.817}
SPL {X  -160.000, Y  +520.912, Z    +0.000, E1   +44.079, E3 +101209.158}
SPL {X  -160.000, Y  +514.086, Z    +0.000, E1   +44.081, E3 +101224.106}
SPL {X  -160.000, Y  +507.208, Z    +0.000, E1   +44.082, E3 +101239.182}
SPL {X  -160.000, Y  +499.184, Z    +0.000, E1   +44.113, E3 +101256.741}
ENDSPLINE

SPLINE
SPL {X  -160.000, Y  +503.824, Z    +0.000, E1   +39.488, E3 +101272.789}
ENDSPLINE

SPLINE
SPL {X  -160.000, Y  +499.279, Z    +0.000, E1   +38.981, E3 +101287.779}
SPL {X  -160.000, Y  +490.068, Z    +0.000, E1   +40.198, E3 +101304.083}
SPL {X  -160.000, Y  +481.368, Z    +0.000, E1   +41.274, E3 +101319.073}
SPL {X  -160.000, Y  +470.910, Z    +0.000, E1   +42.658, E3 +101335.582}
SPL {X  -160.000, Y  +460.219, Z    +0.000, E1   +43.912, E3 +101352.202}
SPL {X  -160.000, Y  +451.951, Z    +0.000, E1   +44.355, E3 +101367.768}
SPL {X  -160.000, Y  +442.331, Z    +0.000, E1   +44.390, E3 +101388.632}
SPL {X  -160.000, Y  +433.037, Z    +0.000, E1   +44.348, E3 +101408.906}
SPL {X  -160.000, Y  +424.435, Z    +0.000, E1   +44.358, E3 +101427.575}
SPL {X  -160.000, Y  +416.015, Z    +0.000, E1   +44.348, E3 +101445.895}
SPL {X  -160.000, Y  +407.167, Z    +0.000, E1   +44.365, E3 +101465.105}
SPL {X  -160.000, Y  +397.599, Z    +0.000, E1   +44.371, E3 +101485.914}
SPL {X  -160.000, Y  +388.533, Z    +0.000, E1   +44.340, E3 +101505.688}
SPL {X  -159.759, Y  +380.021, Z    +0.000, E1   +44.311, E3 +101524.421}
SPL {X  -159.014, Y  +371.065, Z    +0.000, E1   +44.193, E3 +101544.659}
SPL {X  -157.745, Y  +362.030, Z    +0.000, E1   +43.965, E3 +101565.641}
SPL {X  -156.258, Y  +354.400, Z    +0.000, E1   +43.653, E3 +101583.848}
SPL {X  -154.385, Y  +346.786, Z    +0.000, E1   +43.356, E3 +101602.260}
SPL {X  -152.146, Y  +339.286, Z    +0.000, E1   +42.904, E3 +101620.894}
SPL {X  -149.854, Y  +332.731, Z    +0.000, E1   +42.474, E3 +101637.422}
SPL {X  -145.635, Y  +322.541, Z    +0.000, E1   +36.397, E3 +101713.381}
ENDSPLINE

SPLINE
SPL {X  -156.682, Y  +356.385, Z    +0.000, E1   +19.033, E3 +101771.687}
SPL {X  -159.526, Y  +376.492, Z    +0.000, E1    +8.067, E3 +101781.596}
SPL {X  -159.961, Y  +385.275, Z    +0.000, E1    +2.550, E3 +101783.635}
SPL {X  -160.000, Y  +390.345, Z    +0.000, E1    -1.188, E3 +101784.361}
SPL {X  -160.000, Y  +395.838, Z    +0.000, E1    -6.211, E3 +101785.304}
SPL {X  -160.000, Y  +403.277, Z    +0.000, E1   -14.057, E3 +101787.255}
SPL {X  -160.000, Y  +414.316, Z    +0.000, E1   -24.810, E3 +101792.328}
SPL {X  -160.000, Y  +442.604, Z    +0.000, E1   -40.161, E3 +101814.462}
SPL {X  -160.000, Y  +482.867, Z    +0.000, E1   -45.148, E3 +101874.679}
SPL {X  -160.000, Y  +494.769, Z    +0.000, E1   -45.151, E3 +101899.898}
SPL {X  -160.000, Y  +505.761, Z    +0.000, E1   -45.118, E3 +101923.212}
SPL {X  -160.000, Y  +517.347, Z    +0.000, E1   -45.173, E3 +101947.649}
SPL {X  -160.000, Y  +529.298, Z    +0.000, E1   -45.138, E3 +101973.033}
SPL {X  -160.000, Y  +540.664, Z    +0.000, E1   -45.139, E3 +101997.111}
SPL {X  -160.000, Y  +552.011, Z    +0.000, E1   -45.139, E3 +102021.147}
SPL {X  -160.000, Y  +563.667, Z    +0.000, E1   -45.146, E3 +102045.827}
SPL {X  -160.000, Y  +574.965, Z    +0.000, E1   -45.125, E3 +102069.803}
SPL {X  -160.000, Y  +585.644, Z    +0.000, E1   -45.117, E3 +102092.443}
SPL {X  -160.000, Y  +596.819, Z    +0.000, E1   -45.144, E3 +102116.084}
SPL {X  -160.000, Y  +608.165, Z    +0.000, E1   -45.120, E3 +102140.159}
SPL {X  -160.000, Y  +619.270, Z    +0.000, E1   -45.132, E3 +102163.661}
SPL {X  -160.000, Y  +629.968, Z    +0.000, E1   -45.117, E3 +102186.327}
SPL {X  -160.000, Y  +640.750, Z    +0.000, E1   -45.131, E3 +102209.150}
SPL {X  -160.000, Y  +651.429, Z    +0.000, E1   -45.117, E3 +102231.792}
SPL {X  -160.000, Y  +662.434, Z    +0.000, E1   -45.129, E3 +102255.136}
SPL {X  -159.992, Y  +673.110, Z    +0.000, E1   -45.097, E3 +102277.828}
SPL {X  -159.521, Y  +683.874, Z    +0.000, E1   -45.054, E3 +102301.083}
SPL {X  -158.435, Y  +693.823, Z    +0.000, E1   -44.810, E3 +102323.388}
SPL {X  -156.807, Y  +703.304, Z    +0.000, E1   -44.558, E3 +102345.108}
SPL {X  -154.802, Y  +711.950, Z    +0.000, E1   -44.141, E3 +102365.568}
SPL {X  -152.641, Y  +719.464, Z    +0.000, E1   -43.749, E3 +102383.684}
SPL {X  -149.826, Y  +727.645, Z    +0.000, E1   -43.252, E3 +102403.787}
SPL {X  -145.307, Y  +738.478, Z    +0.000, E1   -36.676, E3 +102483.855}
ENDSPLINE

SPLINE
SPL {X  -155.601, Y  +708.762, Z    +0.000, E1   -21.463, E3 +102538.641}
SPL {X  -158.549, Y  +693.002, Z    +0.000, E1   -13.406, E3 +102547.632}
SPL {X  -159.716, Y  +681.031, Z    +0.000, E1    -6.529, E3 +102551.782}
SPL {X  -160.000, Y  +671.641, Z    +0.000, E1    -0.547, E3 +102553.499}
SPL {X  -160.000, Y  +665.424, Z    +0.000, E1    +5.044, E3 +102554.447}
SPL {X  -160.000, Y  +658.015, Z    +0.000, E1   +12.630, E3 +102556.365}
SPL {X  -160.000, Y  +645.110, Z    +0.000, E1   +25.142, E3 +102562.165}
SPL {X  -160.000, Y  +611.664, Z    +0.000, E1   +41.262, E3 +102591.894}
SPL {X  -160.000, Y  +581.433, Z    +0.000, E1   +44.103, E3 +102641.631}
SPL {X  -160.000, Y  +572.090, Z    +0.000, E1   +44.120, E3 +102662.095}
SPL {X  -160.000, Y  +563.431, Z    +0.000, E1   +44.084, E3 +102681.149}
SPL {X  -160.000, Y  +556.107, Z    +0.000, E1   +44.076, E3 +102697.217}
SPL {X  -160.000, Y  +549.181, Z    +0.000, E1   +44.079, E3 +102712.377}
SPL {X  -160.000, Y  +542.413, Z    +0.000, E1   +44.088, E3 +102727.211}
SPL {X  -160.000, Y  +534.609, Z    +0.000, E1   +44.095, E3 +102744.321}
SPL {X  -160.000, Y  +527.457, Z    +0.000, E1   +44.070, E3 +102760.031}
SPL {X  -160.000, Y  +520.912, Z    +0.000, E1   +44.079, E3 +102774.372}
SPL {X  -160.000, Y  +514.086, Z    +0.000, E1   +44.081, E3 +102789.320}
SPL {X  -160.000, Y  +507.208, Z    +0.000, E1   +44.082, E3 +102804.397}
SPL {X  -160.000, Y  +499.184, Z    +0.000, E1   +44.113, E3 +102821.955}
ENDSPLINE

SPLINE
SPL {X  -160.000, Y  +503.824, Z    +0.000, E1   +39.488, E3 +102838.003}
ENDSPLINE

SPLINE
SPL {X  -160.000, Y  +499.279, Z    +0.000, E1   +38.981, E3 +102852.993}
SPL {X  -160.000, Y  +490.068, Z    +0.000, E1   +40.198, E3 +102869.297}
SPL {X  -160.000, Y  +481.368, Z    +0.000, E1   +41.274, E3 +102884.287}
SPL {X  -160.000, Y  +470.910, Z    +0.000, E1   +42.658, E3 +102900.796}
SPL {X  -160.000, Y  +460.219, Z    +0.000, E1   +43.912, E3 +102917.417}
SPL {X  -160.000, Y  +451.951, Z    +0.000, E1   +44.355, E3 +102932.982}
SPL {X  -160.000, Y  +442.331, Z    +0.000, E1   +44.390, E3 +102953.846}
SPL {X  -160.000, Y  +433.037, Z    +0.000, E1   +44.348, E3 +102974.120}
SPL {X  -160.000, Y  +424.435, Z    +0.000, E1   +44.358, E3 +102992.789}
SPL {X  -160.000, Y  +416.015, Z    +0.000, E1   +44.348, E3 +103011.109}
SPL {X  -160.000, Y  +407.167, Z    +0.000, E1   +44.365, E3 +103030.319}
SPL {X  -160.000, Y  +397.599, Z    +0.000, E1   +44.371, E3 +103051.128}
SPL {X  -160.000, Y  +388.533, Z    +0.000, E1   +44.340, E3 +103070.903}
SPL {X  -159.759, Y  +380.021, Z    +0.000, E1   +44.311, E3 +103089.635}
SPL {X  -159.014, Y  +371.065, Z    +0.000, E1   +44.193, E3 +103109.873}
SPL {X  -157.745, Y  +362.030, Z    +0.000, E1   +43.965, E3 +103130.855}
SPL {X  -156.258, Y  +354.400, Z    +0.000, E1   +43.653, E3 +103149.062}
SPL {X  -154.385, Y  +346.786, Z    +0.000, E1   +43.356, E3 +103167.474}
SPL {X  -152.146, Y  +339.286, Z    +0.000, E1   +42.904, E3 +103186.108}
SPL {X  -149.854, Y  +332.731, Z    +0.000, E1   +42.474, E3 +103202.636}
SPL {X  -145.635, Y  +322.541, Z    +0.000, E1   +36.397, E3 +103278.595}
ENDSPLINE

SPLINE
SPL {X  -156.682, Y  +356.385, Z    +0.000, E1   +19.033, E3 +103336.901}
SPL {X  -159.526, Y  +376.492, Z    +0.000, E1    +8.067, E3 +103346.810}
SPL {X  -159.961, Y  +385.275, Z    +0.000, E1    +2.550, E3 +103348.849}
SPL {X  -160.000, Y  +390.345, Z    +0.000, E1    -1.188, E3 +103349.575}
SPL {X  -160.000, Y  +395.838, Z    +0.000, E1    -6.211, E3 +103350.518}
SPL {X  -160.000, Y  +403.277, Z    +0.000, E1   -14.057, E3 +103352.469}
SPL {X  -160.000, Y  +414.316, Z    +0.000, E1   -24.810, E3 +103357.542}
SPL {X  -160.000, Y  +442.604, Z    +0.000, E1   -40.161, E3 +103379.677}
SPL {X  -160.000, Y  +482.867, Z    +0.000, E1   -45.148, E3 +103439.893}
SPL {X  -160.000, Y  +494.769, Z    +0.000, E1   -45.151, E3 +103465.112}
SPL {X  -160.000, Y  +505.761, Z    +0.000, E1   -45.118, E3 +103488.426}
SPL {X  -160.000, Y  +517.347, Z    +0.000, E1   -45.173, E3 +103512.864}
SPL {X  -160.000, Y  +529.298, Z    +0.000, E1   -45.138, E3 +103538.247}
SPL {X  -160.000, Y  +540.664, Z    +0.000, E1   -45.139, E3 +103562.325}
SPL {X  -160.000, Y  +552.011, Z    +0.000, E1   -45.139, E3 +103586.361}
SPL {X  -160.000, Y  +563.667, Z    +0.000, E1   -45.146, E3 +103611.041}
SPL {X  -160.000, Y  +574.965, Z    +0.000, E1   -45.125, E3 +103635.017}
SPL {X  -160.000, Y  +585.644, Z    +0.000, E1   -45.117, E3 +103657.657}
SPL {X  -160.000, Y  +596.819, Z    +0.000, E1   -45.144, E3 +103681.298}
SPL {X  -160.000, Y  +608.165, Z    +0.000, E1   -45.120, E3 +103705.373}
SPL {X  -160.000, Y  +619.270, Z    +0.000, E1   -45.132, E3 +103728.875}
SPL {X  -160.000, Y  +629.968, Z    +0.000, E1   -45.117, E3 +103751.542}
SPL {X  -160.000, Y  +640.750, Z    +0.000, E1   -45.131, E3 +103774.365}
SPL {X  -160.000, Y  +651.429, Z    +0.000, E1   -45.117, E3 +103797.006}
SPL {X  -160.000, Y  +662.434, Z    +0.000, E1   -45.129, E3 +103820.350}
SPL {X  -159.992, Y  +673.110, Z    +0.000, E1   -45.097, E3 +103843.042}
SPL {X  -159.521, Y  +683.874, Z    +0.000, E1   -45.054, E3 +103866.298}
SPL {X  -158.435, Y  +693.823, Z    +0.000, E1   -44.810, E3 +103888.602}
SPL {X  -156.807, Y  +703.304, Z    +0.000, E1   -44.558, E3 +103910.323}
SPL {X  -154.802, Y  +711.950, Z    +0.000, E1   -44.141, E3 +103930.783}
SPL {X  -152.641, Y  +719.464, Z    +0.000, E1   -43.749, E3 +103948.898}
SPL {X  -149.826, Y  +727.645, Z    +0.000, E1   -43.252, E3 +103969.001}
SPL {X  -145.307, Y  +738.478, Z    +0.000, E1   -36.676, E3 +104049.069}
ENDSPLINE

SPLINE
SPL {X  -155.601, Y  +708.762, Z    +0.000, E1   -21.463, E3 +104103.856}
SPL {X  -158.549, Y  +693.002, Z    +0.000, E1   -13.406, E3 +104112.846}
SPL {X  -159.716, Y  +681.031, Z    +0.000, E1    -6.529, E3 +104116.996}
SPL {X  -160.000, Y  +671.641, Z    +0.000, E1    -0.547, E3 +104118.713}
SPL {X  -160.000, Y  +665.424, Z    +0.000, E1    +5.044, E3 +104119.661}
SPL {X  -160.000, Y  +658.015, Z    +0.000, E1   +12.630, E3 +104121.579}
SPL {X  -160.000, Y  +645.110, Z    +0.000, E1   +25.142, E3 +104127.379}
SPL {X  -160.000, Y  +611.664, Z    +0.000, E1   +41.262, E3 +104157.108}
SPL {X  -160.000, Y  +581.433, Z    +0.000, E1   +44.103, E3 +104206.845}
SPL {X  -160.000, Y  +572.090, Z    +0.000, E1   +44.120, E3 +104227.310}
SPL {X  -160.000, Y  +563.431, Z    +0.000, E1   +44.084, E3 +104246.363}
SPL {X  -160.000, Y  +556.107, Z    +0.000, E1   +44.076, E3 +104262.431}
SPL {X  -160.000, Y  +549.181, Z    +0.000, E1   +44.079, E3 +104277.591}
SPL {X  -160.000, Y  +542.413, Z    +0.000, E1   +44.088, E3 +104292.425}
SPL {X  -160.000, Y  +534.609, Z    +0.000, E1   +44.095, E3 +104309.535}
SPL {X  -160.000, Y  +527.457, Z    +0.000, E1   +44.070, E3 +104325.245}
SPL {X  -160.000, Y  +520.912, Z    +0.000, E1   +44.079, E3 +104339.586}
SPL {X  -160.000, Y  +514.086, Z    +0.000, E1   +44.081, E3 +104354.534}
SPL {X  -160.000, Y  +507.208, Z    +0.000, E1   +44.082, E3 +104369.611}
SPL {X  -160.000, Y  +499.184, Z    +0.000, E1   +44.113, E3 +104387.169}
ENDSPLINE

SPLINE
SPL {X  -160.000, Y  +503.824, Z    +0.000, E1   +39.488, E3 +104403.218}
ENDSPLINE

SPLINE
SPL {X  -160.000, Y  +499.279, Z    +0.000, E1   +38.981, E3 +104418.208}
SPL {X  -160.000, Y  +490.068, Z    +0.000, E1   +40.198, E3 +104434.512}
SPL {X  -160.000, Y  +481.368, Z    +0.000, E1   +41.274, E3 +104449.501}
SPL {X  -160.000, Y  +470.910, Z    +0.000, E1   +42.658, E3 +104466.010}
SPL {X  -160.000, Y  +460.219, Z    +0.000, E1   +43.912, E3 +104482.631}
SPL {X  -160.000, Y  +451.951, Z    +0.000, E1   +44.355, E3 +104498.196}
SPL {X  -160.000, Y  +442.331, Z    +0.000, E1   +44.390, E3 +104519.060}
SPL {X  -160.000, Y  +433.037, Z    +0.000, E1   +44.348, E3 +104539.334}
SPL {X  -160.000, Y  +424.435, Z    +0.000, E1   +44.358, E3 +104558.003}
SPL {X  -160.000, Y  +416.015, Z    +0.000, E1   +44.348, E3 +104576.323}
SPL {X  -160.000, Y  +407.167, Z    +0.000, E1   +44.365, E3 +104595.534}
SPL {X  -160.000, Y  +397.599, Z    +0.000, E1   +44.371, E3 +104616.342}
SPL {X  -160.000, Y  +388.533, Z    +0.000, E1   +44.340, E3 +104636.117}
SPL {X  -159.759, Y  +380.021, Z    +0.000, E1   +44.311, E3 +104654.849}
SPL {X  -159.014, Y  +371.065, Z    +0.000, E1   +44.193, E3 +104675.087}
SPL {X  -157.745, Y  +362.030, Z    +0.000, E1   +43.965, E3 +104696.069}
SPL {X  -156.258, Y  +354.400, Z    +0.000, E1   +43.653, E3 +104714.276}
SPL {X  -154.385, Y  +346.786, Z    +0.000, E1   +43.356, E3 +104732.688}
SPL {X  -152.146, Y  +339.286, Z    +0.000, E1   +42.904, E3 +104751.323}
SPL {X  -149.854, Y  +332.731, Z    +0.000, E1   +42.474, E3 +104767.850}
SPL {X  -145.635, Y  +322.541, Z    +0.000, E1   +36.397, E3 +104843.809}
ENDSPLINE

SPLINE
SPL {X  -156.682, Y  +356.385, Z    +0.000, E1   +19.033, E3 +104902.115}
SPL {X  -159.526, Y  +376.492, Z    +0.000, E1    +8.067, E3 +104912.025}
SPL {X  -159.961, Y  +385.275, Z    +0.000, E1    +2.550, E3 +104914.063}
SPL {X  -160.000, Y  +390.345, Z    +0.000, E1    -1.188, E3 +104914.789}
SPL {X  -160.000, Y  +395.838, Z    +0.000, E1    -6.211, E3 +104915.732}
SPL {X  -160.000, Y  +403.277, Z    +0.000, E1   -14.057, E3 +104917.684}
SPL {X  -160.000, Y  +414.316, Z    +0.000, E1   -24.810, E3 +104922.757}
SPL {X  -160.000, Y  +442.604, Z    +0.000, E1   -40.161, E3 +104944.891}
SPL {X  -160.000, Y  +482.867, Z    +0.000, E1   -45.148, E3 +105005.107}
SPL {X  -160.000, Y  +494.769, Z    +0.000, E1   -45.151, E3 +105030.326}
SPL {X  -160.000, Y  +505.761, Z    +0.000, E1   -45.118, E3 +105053.640}
SPL {X  -160.000, Y  +517.347, Z    +0.000, E1   -45.173, E3 +105078.078}
SPL {X  -160.000, Y  +529.298, Z    +0.000, E1   -45.138, E3 +105103.461}
SPL {X  -160.000, Y  +540.664, Z    +0.000, E1   -45.139, E3 +105127.539}
SPL {X  -160.000, Y  +552.011, Z    +0.000, E1   -45.139, E3 +105151.575}
SPL {X  -160.000, Y  +563.667, Z    +0.000, E1   -45.146, E3 +105176.255}
SPL {X  -160.000, Y  +574.965, Z    +0.000, E1   -45.125, E3 +105200.231}
SPL {X  -160.000, Y  +585.644, Z    +0.000, E1   -45.117, E3 +105222.871}
SPL {X  -160.000, Y  +596.819, Z    +0.000, E1   -45.144, E3 +105246.513}
SPL {X  -160.000, Y  +608.165, Z    +0.000, E1   -45.120, E3 +105270.587}
SPL {X  -160.000, Y  +619.270, Z    +0.000, E1   -45.132, E3 +105294.089}
SPL {X  -160.000, Y  +629.968, Z    +0.000, E1   -45.117, E3 +105316.756}
SPL {X  -160.000, Y  +640.750, Z    +0.000, E1   -45.131, E3 +105339.579}
SPL {X  -160.000, Y  +651.429, Z    +0.000, E1   -45.117, E3 +105362.220}
SPL {X  -160.000, Y  +662.434, Z    +0.000, E1   -45.129, E3 +105385.564}
SPL {X  -159.992, Y  +673.110, Z    +0.000, E1   -45.097, E3 +105408.257}
SPL {X  -159.521, Y  +683.874, Z    +0.000, E1   -45.054, E3 +105431.512}
SPL {X  -158.435, Y  +693.823, Z    +0.000, E1   -44.810, E3 +105453.816}
SPL {X  -156.807, Y  +703.304, Z    +0.000, E1   -44.558, E3 +105475.537}
SPL {X  -154.802, Y  +711.950, Z    +0.000, E1   -44.141, E3 +105495.997}
SPL {X  -152.641, Y  +719.464, Z    +0.000, E1   -43.749, E3 +105514.113}
SPL {X  -149.826, Y  +727.645, Z    +0.000, E1   -43.252, E3 +105534.215}
SPL {X  -145.307, Y  +738.478, Z    +0.000, E1   -36.676, E3 +105614.283}
ENDSPLINE

SPLINE
SPL {X  -155.601, Y  +708.762, Z    +0.000, E1   -21.463, E3 +105669.070}
SPL {X  -158.549, Y  +693.002, Z    +0.000, E1   -13.406, E3 +105678.060}
SPL {X  -159.716, Y  +681.031, Z    +0.000, E1    -6.529, E3 +105682.211}
SPL {X  -160.000, Y  +671.641, Z    +0.000, E1    -0.547, E3 +105683.927}
SPL {X  -160.000, Y  +665.424, Z    +0.000, E1    +5.044, E3 +105684.875}
SPL {X  -160.000, Y  +658.015, Z    +0.000, E1   +12.630, E3 +105686.793}
SPL {X  -160.000, Y  +645.110, Z    +0.000, E1   +25.142, E3 +105692.593}
SPL {X  -160.000, Y  +611.664, Z    +0.000, E1   +41.262, E3 +105722.323}
SPL {X  -160.000, Y  +581.433, Z    +0.000, E1   +44.103, E3 +105772.059}
SPL {X  -160.000, Y  +572.090, Z    +0.000, E1   +44.120, E3 +105792.524}
SPL {X  -160.000, Y  +563.431, Z    +0.000, E1   +44.084, E3 +105811.577}
SPL {X  -160.000, Y  +556.107, Z    +0.000, E1   +44.076, E3 +105827.645}
SPL {X  -160.000, Y  +549.181, Z    +0.000, E1   +44.079, E3 +105842.805}
SPL {X  -160.000, Y  +542.413, Z    +0.000, E1   +44.088, E3 +105857.639}
SPL {X  -160.000, Y  +534.609, Z    +0.000, E1   +44.095, E3 +105874.749}
SPL {X  -160.000, Y  +527.457, Z    +0.000, E1   +44.070, E3 +105890.459}
SPL {X  -160.000, Y  +520.912, Z    +0.000, E1   +44.079, E3 +105904.800}
SPL {X  -160.000, Y  +514.086, Z    +0.000, E1   +44.081, E3 +105919.748}
SPL {X  -160.000, Y  +507.208, Z    +0.000, E1   +44.082, E3 +105934.825}
SPL {X  -160.000, Y  +499.184, Z    +0.000, E1   +44.113, E3 +105952.383}
ENDSPLINE

SPLINE
SPL {X  -160.000, Y  +503.824, Z    +0.000, E1   +39.488, E3 +105968.432}
ENDSPLINE

SPLINE
SPL {X  -160.000, Y  +499.279, Z    +0.000, E1   +38.981, E3 +105983.422}
SPL {X  -160.000, Y  +490.068, Z    +0.000, E1   +40.198, E3 +105999.726}
SPL {X  -160.000, Y  +481.368, Z    +0.000, E1   +41.274, E3 +106014.716}
SPL {X  -160.000, Y  +470.910, Z    +0.000, E1   +42.658, E3 +106031.224}
SPL {X  -160.000, Y  +460.219, Z    +0.000, E1   +43.912, E3 +106047.845}
SPL {X  -160.000, Y  +451.951, Z    +0.000, E1   +44.355, E3 +106063.410}
SPL {X  -160.000, Y  +442.331, Z    +0.000, E1   +44.390, E3 +106084.275}
SPL {X  -160.000, Y  +433.037, Z    +0.000, E1   +44.348, E3 +106104.549}
SPL {X  -160.000, Y  +424.435, Z    +0.000, E1   +44.358, E3 +106123.217}
SPL {X  -160.000, Y  +416.015, Z    +0.000, E1   +44.348, E3 +106141.537}
SPL {X  -160.000, Y  +407.167, Z    +0.000, E1   +44.365, E3 +106160.748}
SPL {X  -160.000, Y  +397.599, Z    +0.000, E1   +44.371, E3 +106181.556}
SPL {X  -160.000, Y  +388.533, Z    +0.000, E1   +44.340, E3 +106201.331}
SPL {X  -159.759, Y  +380.021, Z    +0.000, E1   +44.311, E3 +106220.063}
SPL {X  -159.014, Y  +371.065, Z    +0.000, E1   +44.193, E3 +106240.301}
SPL {X  -157.745, Y  +362.030, Z    +0.000, E1   +43.965, E3 +106261.283}
SPL {X  -156.258, Y  +354.400, Z    +0.000, E1   +43.653, E3 +106279.490}
SPL {X  -154.385, Y  +346.786, Z    +0.000, E1   +43.356, E3 +106297.902}
SPL {X  -152.146, Y  +339.286, Z    +0.000, E1   +42.904, E3 +106316.537}
SPL {X  -149.854, Y  +332.731, Z    +0.000, E1   +42.474, E3 +106333.065}
SPL {X  -145.635, Y  +322.541, Z    +0.000, E1   +36.397, E3 +106409.024}
ENDSPLINE

SPLINE
SPL {X  -156.682, Y  +356.385, Z    +0.000, E1   +19.033, E3 +106467.330}
SPL {X  -159.526, Y  +376.492, Z    +0.000, E1    +8.067, E3 +106477.239}
SPL {X  -159.961, Y  +385.275, Z    +0.000, E1    +2.550, E3 +106479.277}
SPL {X  -160.000, Y  +390.345, Z    +0.000, E1    -1.188, E3 +106480.003}
SPL {X  -160.000, Y  +395.838, Z    +0.000, E1    -6.211, E3 +106480.947}
SPL {X  -160.000, Y  +403.277, Z    +0.000, E1   -14.057, E3 +106482.898}
SPL {X  -160.000, Y  +414.316, Z    +0.000, E1   -24.810, E3 +106487.971}
SPL {X  -160.000, Y  +442.604, Z    +0.000, E1   -40.161, E3 +106510.105}
SPL {X  -160.000, Y  +482.867, Z    +0.000, E1   -45.148, E3 +106570.321}
SPL {X  -160.000, Y  +494.769, Z    +0.000, E1   -45.151, E3 +106595.540}
SPL {X  -160.000, Y  +505.761, Z    +0.000, E1   -45.118, E3 +106618.854}
SPL {X  -160.000, Y  +517.347, Z    +0.000, E1   -45.173, E3 +106643.292}
SPL {X  -160.000, Y  +529.298, Z    +0.000, E1   -45.138, E3 +106668.675}
SPL {X  -160.000, Y  +540.664, Z    +0.000, E1   -45.139, E3 +106692.753}
SPL {X  -160.000, Y  +552.011, Z    +0.000, E1   -45.139, E3 +106716.789}
SPL {X  -160.000, Y  +563.667, Z    +0.000, E1   -45.146, E3 +106741.469}
SPL {X  -160.000, Y  +574.965, Z    +0.000, E1   -45.125, E3 +106765.445}
SPL {X  -160.000, Y  +585.644, Z    +0.000, E1   -45.117, E3 +106788.085}
SPL {X  -160.000, Y  +596.819, Z    +0.000, E1   -45.144, E3 +106811.727}
SPL {X  -160.000, Y  +608.165, Z    +0.000, E1   -45.120, E3 +106835.801}
SPL {X  -160.000, Y  +619.270, Z    +0.000, E1   -45.132, E3 +106859.304}
SPL {X  -160.000, Y  +629.968, Z    +0.000, E1   -45.117, E3 +106881.970}
SPL {X  -160.000, Y  +640.750, Z    +0.000, E1   -45.131, E3 +106904.793}
SPL {X  -160.000, Y  +651.429, Z    +0.000, E1   -45.117, E3 +106927.434}
SPL {X  -160.000, Y  +662.434, Z    +0.000, E1   -45.129, E3 +106950.778}
SPL {X  -159.992, Y  +673.110, Z    +0.000, E1   -45.097, E3 +106973.471}
SPL {X  -159.521, Y  +683.874, Z    +0.000, E1   -45.054, E3 +106996.726}
SPL {X  -158.435, Y  +693.823, Z    +0.000, E1   -44.810, E3 +107019.030}
SPL {X  -156.807, Y  +703.304, Z    +0.000, E1   -44.558, E3 +107040.751}
SPL {X  -154.802, Y  +711.950, Z    +0.000, E1   -44.141, E3 +107061.211}
SPL {X  -152.641, Y  +719.464, Z    +0.000, E1   -43.749, E3 +107079.327}
SPL {X  -149.826, Y  +727.645, Z    +0.000, E1   -43.252, E3 +107099.430}
SPL {X  -145.307, Y  +738.478, Z    +0.000, E1   -36.676, E3 +107179.497}
ENDSPLINE

SPLINE
SPL {X  -155.601, Y  +708.762, Z    +0.000, E1   -21.463, E3 +107234.284}
SPL {X  -158.549, Y  +693.002, Z    +0.000, E1   -13.406, E3 +107243.275}
SPL {X  -159.716, Y  +681.031, Z    +0.000, E1    -6.529, E3 +107247.425}
SPL {X  -160.000, Y  +671.641, Z    +0.000, E1    -0.547, E3 +107249.141}
SPL {X  -160.000, Y  +665.424, Z    +0.000, E1    +5.044, E3 +107250.090}
SPL {X  -160.000, Y  +658.015, Z    +0.000, E1   +12.630, E3 +107252.007}
SPL {X  -160.000, Y  +645.110, Z    +0.000, E1   +25.142, E3 +107257.807}
SPL {X  -160.000, Y  +611.664, Z    +0.000, E1   +41.262, E3 +107287.537}
SPL {X  -160.000, Y  +581.433, Z    +0.000, E1   +44.103, E3 +107337.274}
SPL {X  -160.000, Y  +572.090, Z    +0.000, E1   +44.120, E3 +107357.738}
SPL {X  -160.000, Y  +563.431, Z    +0.000, E1   +44.084, E3 +107376.791}
SPL {X  -160.000, Y  +556.107, Z    +0.000, E1   +44.076, E3 +107392.859}
SPL {X  -160.000, Y  +549.181, Z    +0.000, E1   +44.079, E3 +107408.019}
SPL {X  -160.000, Y  +542.413, Z    +0.000, E1   +44.088, E3 +107422.853}
SPL {X  -160.000, Y  +534.609, Z    +0.000, E1   +44.095, E3 +107439.963}
SPL {X  -160.000, Y  +527.457, Z    +0.000, E1   +44.070, E3 +107455.673}
SPL {X  -160.000, Y  +520.912, Z    +0.000, E1   +44.079, E3 +107470.014}
SPL {X  -160.000, Y  +514.086, Z    +0.000, E1   +44.081, E3 +107484.963}
SPL {X  -160.000, Y  +507.208, Z    +0.000, E1   +44.082, E3 +107500.039}
SPL {X  -160.000, Y  +499.184, Z    +0.000, E1   +44.113, E3 +107517.597}
ENDSPLINE

SPLINE
SPL {X  -160.000, Y  +503.824, Z    +0.000, E1   +39.488, E3 +107533.646}
ENDSPLINE

SPLINE
SPL {X  -160.000, Y  +499.279, Z    +0.000, E1   +38.981, E3 +107548.636}
SPL {X  -160.000, Y  +490.068, Z    +0.000, E1   +40.198, E3 +107564.940}
SPL {X  -160.000, Y  +481.368, Z    +0.000, E1   +41.274, E3 +107579.930}
SPL {X  -160.000, Y  +470.910, Z    +0.000, E1   +42.658, E3 +107596.438}
SPL {X  -160.000, Y  +460.218, Z    +0.000, E1   +43.912, E3 +107613.059}
ENDSPLINE
=
SPLINE
SPL {X  -160.000, Y  +465.362, Z    +0.000, E1   +38.803, E3 +107631.994}
SPL {X  -160.000, Y  +457.266, Z    +0.000, E1   +38.756, E3 +107653.503}
SPL {X  -160.000, Y  +448.553, Z    +0.000, E1   +38.823, E3 +107676.454}
SPL {X  -160.000, Y  +439.425, Z    +0.000, E1   +38.797, E3 +107700.625}
SPL {X  -160.000, Y  +430.351, Z    +0.000, E1   +38.810, E3 +107724.640}
SPL {X  -160.000, Y  +421.477, Z    +0.000, E1   +38.792, E3 +107748.143}
SPL {X  -160.000, Y  +412.292, Z    +0.000, E1   +38.825, E3 +107772.371}
SPL {X  -160.000, Y  +403.281, Z    +0.000, E1   +38.797, E3 +107796.251}
SPL {X  -160.000, Y  +394.948, Z    +0.000, E1   +38.796, E3 +107818.292}
SPL {X  -159.971, Y  +385.741, Z    +0.000, E1   +38.831, E3 +107842.614}
SPL {X  -159.525, Y  +376.478, Z    +0.000, E1   +38.739, E3 +107867.605}
SPL {X  -158.721, Y  +368.613, Z    +0.000, E1   +38.561, E3 +107889.328}
SPL {X  -157.505, Y  +360.654, Z    +0.000, E1   +38.390, E3 +107911.601}
SPL {X  -156.229, Y  +354.269, Z    +0.000, E1   +38.076, E3 +107929.951}
SPL {X  -155.202, Y  +349.910, Z    +0.000, E1   +37.893, E3 +107942.525}
SPL {X  -154.128, Y  +345.852, Z    +0.000, E1   +37.701, E3 +107954.349}
SPL {X  -152.890, Y  +341.633, Z    +0.000, E1   +37.487, E3 +107966.781}
SPL {X  -150.284, Y  +333.893, Z    +0.000, E1   +33.433, E3 +108021.592}
ENDSPLINE

SPLINE
SPL {X  -157.404, Y  +360.095, Z    +0.000, E1   +17.695, E3 +108076.716}
SPL {X  -159.413, Y  +375.108, Z    +0.000, E1    +9.284, E3 +108085.805}
SPL {X  -159.978, Y  +386.135, Z    +0.000, E1    +2.544, E3 +108089.366}
SPL {X  -160.000, Y  +393.708, Z    +0.000, E1    -3.216, E3 +108091.120}
SPL {X  -160.000, Y  +400.474, Z    +0.000, E1    -9.529, E3 +108093.167}
SPL {X  -160.000, Y  +409.652, Z    +0.000, E1   -18.026, E3 +108097.303}
SPL {X  -160.000, Y  +437.804, Z    +0.000, E1   -34.779, E3 +108122.096}
SPL {X  -160.000, Y  +463.067, Z    +0.000, E1   -38.672, E3 +108167.796}
SPL {X  -160.000, Y  +469.167, Z    +0.000, E1   -38.717, E3 +108183.902}
SPL {X  -160.000, Y  +476.691, Z    +0.000, E1   -38.728, E3 +108203.834}
SPL {X  -160.000, Y  +483.419, Z    +0.000, E1   -38.692, E3 +108221.734}
SPL {X  -160.000, Y  +489.013, Z    +0.000, E1   -38.683, E3 +108236.573}
SPL {X  -160.000, Y  +494.786, Z    +0.000, E1   -38.693, E3 +108251.883}
SPL {X  -160.000, Y  +500.108, Z    +0.000, E1   -38.668, E3 +108266.034}
SPL {X  -160.000, Y  +504.903, Z    +0.000, E1   -38.673, E3 +108278.755}
SPL {X  -160.000, Y  +510.180, Z    +0.000, E1   -38.675, E3 +108292.760}
SPL {X  -160.000, Y  +515.083, Z    +0.000, E1   -38.662, E3 +108305.779}
SPL {X  -160.000, Y  +520.479, Z    +0.000, E1   -38.692, E3 +108320.054}
SPL {X  -160.000, Y  +525.998, Z    +0.000, E1   -38.666, E3 +108334.732}
SPL {X  -160.000, Y  +531.341, Z    +0.000, E1   -38.684, E3 +108348.876}
SPL {X  -160.000, Y  +537.313, Z    +0.000, E1   -38.686, E3 +108364.716}
SPL {X  -160.000, Y  +543.203, Z    +0.000, E1   -38.679, E3 +108380.341}
SPL {X  -160.000, Y  +551.201, Z    +0.000, E1   -38.768, E3 +108401.403}
SPL {X  -160.000, Y  +561.335, Z    +0.000, E1   -38.777, E3 +108428.273}
SPL {X  -160.000, Y  +568.812, Z    +0.000, E1   -38.671, E3 +108448.276}
SPL {X  -160.000, Y  +574.116, Z    +0.000, E1   -38.680, E3 +108462.347}
SPL {X  -160.000, Y  +582.193, Z    +0.000, E1   -38.759, E3 +108483.650}
SPL {X  -160.000, Y  +591.932, Z    +0.000, E1   -38.763, E3 +108509.475}
SPL {X  -160.000, Y  +601.488, Z    +0.000, E1   -38.747, E3 +108534.850}
SPL {X  -160.000, Y  +609.161, Z    +0.000, E1   -38.685, E3 +108555.302}
SPL {X  -160.000, Y  +614.445, Z    +0.000, E1   -38.661, E3 +108569.351}
SPL {X  -160.000, Y  +621.895, Z    +0.000, E1   -38.769, E3 +108588.940}
SPL {X  -160.000, Y  +631.692, Z    +0.000, E1   -38.748, E3 +108614.993}
SPL {X  -160.000, Y  +639.246, Z    +0.000, E1   -38.671, E3 +108635.168}
SPL {X  -160.000, Y  +644.827, Z    +0.000, E1   -38.662, E3 +108650.003}
SPL {X  -160.000, Y  +650.491, Z    +0.000, E1   -38.673, E3 +108664.991}
SPL {X  -160.000, Y  +656.011, Z    +0.000, E1   -38.669, E3 +108679.644}
SPL {X  -160.000, Y  +661.156, Z    +0.000, E1   -38.659, E3 +108693.319}
SPL {X  -160.000, Y  +666.701, Z    +0.000, E1   -38.683, E3 +108707.979}
SPL {X  -159.961, Y  +675.011, Z    +0.000, E1   -38.755, E3 +108729.965}
SPL {X  -159.451, Y  +684.743, Z    +0.000, E1   -38.666, E3 +108756.319}
SPL {X  -158.386, Y  +694.170, Z    +0.000, E1   -38.484, E3 +108782.437}
SPL {X  -157.286, Y  +700.846, Z    +0.000, E1   -38.194, E3 +108801.405}
SPL {X  -156.328, Y  +705.580, Z    +0.000, E1   -38.037, E3 +108814.941}
SPL {X  -155.162, Y  +710.549, Z    +0.000, E1   -37.822, E3 +108829.345}
SPL {X  -153.914, Y  +715.210, Z    +0.000, E1   -37.596, E3 +108842.994}
SPL {X  -152.686, Y  +719.322, Z    +0.000, E1   -37.361, E3 +108855.167}
SPL {X  -150.251, Y  +726.496, Z    +0.000, E1   -33.848, E3 +108903.662}
ENDSPLINE

SPLINE
SPL {X  -156.089, Y  +706.662, Z    +0.000, E1   -21.279, E3 +108956.316}
SPL {X  -159.059, Y  +688.824, Z    +0.000, E1   -11.551, E3 +108970.276}
SPL {X  -159.959, Y  +675.119, Z    +0.000, E1    -3.373, E3 +108975.104}
SPL {X  -160.000, Y  +666.447, Z    +0.000, E1    +3.005, E3 +108977.139}
SPL {X  -160.000, Y  +658.774, Z    +0.000, E1   +10.317, E3 +108979.398}
SPL {X  -160.000, Y  +647.765, Z    +0.000, E1   +20.359, E3 +108984.763}
SPL {X  -160.000, Y  +622.607, Z    +0.000, E1   +34.692, E3 +109007.630}
SPL {X  -160.000, Y  +596.106, Z    +0.000, E1   +39.718, E3 +109049.630}
SPL {X  -160.000, Y  +592.273, Z    +0.000, E1   +39.746, E3 +109059.368}
SPL {X  -160.000, Y  +586.287, Z    +0.000, E1   +39.762, E3 +109074.627}
SPL {X  -160.000, Y  +577.753, Z    +0.000, E1   +39.844, E3 +109096.269}
SPL {X  -160.000, Y  +567.367, Z    +0.000, E1   +39.853, E3 +109122.763}
SPL {X  -160.000, Y  +559.466, Z    +0.000, E1   +39.761, E3 +109143.044}
SPL {X  -160.000, Y  +552.914, Z    +0.000, E1   +39.787, E3 +109159.712}
SPL {X  -160.000, Y  +546.390, Z    +0.000, E1   +39.760, E3 +109176.425}
SPL {X  -160.000, Y  +540.123, Z    +0.000, E1   +39.770, E3 +109192.405}
SPL {X  -160.000, Y  +533.658, Z    +0.000, E1   +39.771, E3 +109208.903}
SPL {X  -160.000, Y  +527.046, Z    +0.000, E1   +39.771, E3 +109225.779}
SPL {X  -160.000, Y  +521.063, Z    +0.000, E1   +39.756, E3 +109241.064}
SPL {X  -160.000, Y  +515.110, Z    +0.000, E1   +39.770, E3 +109256.236}
SPL {X  -160.000, Y  +508.717, Z    +0.000, E1   +39.766, E3 +109272.555}
SPL {X  -160.000, Y  +502.133, Z    +0.000, E1   +39.780, E3 +109289.321}
ENDSPLINE

SPLINE
SPL {X  -160.000, Y  +512.949, Z    +0.000, E1   +32.050, E3 +109305.578}
ENDSPLINE

SPLINE
SPL {X  -160.000, Y  +507.092, Z    +0.000, E1   +32.805, E3 +109320.207}
SPL {X  -160.000, Y  +499.824, Z    +0.000, E1   +34.003, E3 +109335.948}
SPL {X  -160.000, Y  +491.367, Z    +0.000, E1   +35.449, E3 +109352.689}
SPL {X  -160.000, Y  +483.082, Z    +0.000, E1   +36.782, E3 +109368.528}
SPL {X  -160.000, Y  +474.521, Z    +0.000, E1   +38.037, E3 +109384.616}
SPL {X  -160.000, Y  +465.343, Z    +0.000, E1   +38.802, E3 +109404.774}
SPL {X  -160.000, Y  +457.266, Z    +0.000, E1   +38.756, E3 +109426.228}
SPL {X  -160.000, Y  +448.553, Z    +0.000, E1   +38.823, E3 +109449.179}
SPL {X  -160.000, Y  +439.425, Z    +0.000, E1   +38.797, E3 +109473.350}
SPL {X  -160.000, Y  +430.351, Z    +0.000, E1   +38.810, E3 +109497.365}
SPL {X  -160.000, Y  +421.477, Z    +0.000, E1   +38.792, E3 +109520.869}
SPL {X  -160.000, Y  +412.292, Z    +0.000, E1   +38.825, E3 +109545.096}
SPL {X  -160.000, Y  +403.281, Z    +0.000, E1   +38.797, E3 +109568.976}
SPL {X  -160.000, Y  +394.948, Z    +0.000, E1   +38.796, E3 +109591.018}
SPL {X  -159.971, Y  +385.741, Z    +0.000, E1   +38.831, E3 +109615.339}
SPL {X  -159.525, Y  +376.478, Z    +0.000, E1   +38.739, E3 +109640.330}
SPL {X  -158.721, Y  +368.613, Z    +0.000, E1   +38.561, E3 +109662.053}
SPL {X  -157.505, Y  +360.654, Z    +0.000, E1   +38.390, E3 +109684.326}
SPL {X  -156.229, Y  +354.269, Z    +0.000, E1   +38.076, E3 +109702.676}
SPL {X  -155.202, Y  +349.910, Z    +0.000, E1   +37.893, E3 +109715.250}
SPL {X  -154.128, Y  +345.852, Z    +0.000, E1   +37.701, E3 +109727.074}
SPL {X  -152.890, Y  +341.633, Z    +0.000, E1   +37.487, E3 +109739.506}
SPL {X  -150.284, Y  +333.893, Z    +0.000, E1   +33.433, E3 +109794.317}
ENDSPLINE

